(* IEC 61131-3 sources: elnaProjects/ElpcLogic/PomarKc7Changed/build_USO_ecl/_ (part 2) *)

  AI_Tstali_statora_kanal_1_HL := ai.Tstali_statora_kanal_1.HL;
  AI_Tstali_statora_kanal_1_LL := ai.Tstali_statora_kanal_1.LL;
  AI_Tstali_statora_kanal_1_status := DWORD_TO_UDINT(ai.Tstali_statora_kanal_1.status);
  AI_Tstali_statora_kanal_1_value := ai.Tstali_statora_kanal_1.value;
  AI_Tstali_statora_kanal_1_HW := ai.Tstali_statora_kanal_1.HW;
  AI_Tstali_statora_kanal_1_newHW := ai.Tstali_statora_kanal_1.dHW;

  AI_Tstali_statora_kanal_2_HL := ai.Tstali_statora_kanal_2.HL;
  AI_Tstali_statora_kanal_2_LL := ai.Tstali_statora_kanal_2.LL;
  AI_Tstali_statora_kanal_2_status := DWORD_TO_UDINT(ai.Tstali_statora_kanal_2.status);
  AI_Tstali_statora_kanal_2_value := ai.Tstali_statora_kanal_2.value;
  AI_Tstali_statora_kanal_2_HW := ai.Tstali_statora_kanal_2.HW;
  AI_Tstali_statora_kanal_2_newHW := ai.Tstali_statora_kanal_2.dHW;

  AI_Tstali_statora_kanal_3_HL := ai.Tstali_statora_kanal_3.HL;
  AI_Tstali_statora_kanal_3_LL := ai.Tstali_statora_kanal_3.LL;
  AI_Tstali_statora_kanal_3_status := DWORD_TO_UDINT(ai.Tstali_statora_kanal_3.status);
  AI_Tstali_statora_kanal_3_value := ai.Tstali_statora_kanal_3.value;
  AI_Tstali_statora_kanal_3_HW := ai.Tstali_statora_kanal_3.HW;
  AI_Tstali_statora_kanal_3_newHW := ai.Tstali_statora_kanal_3.dHW;

  AI_Tmedi_statora_kanal_1_HL := ai.Tmedi_statora_kanal_1.HL;
  AI_Tmedi_statora_kanal_1_LL := ai.Tmedi_statora_kanal_1.LL;
  AI_Tmedi_statora_kanal_1_status := DWORD_TO_UDINT(ai.Tmedi_statora_kanal_1.status);
  AI_Tmedi_statora_kanal_1_value := ai.Tmedi_statora_kanal_1.value;
  AI_Tmedi_statora_kanal_1_HW := ai.Tmedi_statora_kanal_1.HW;
  AI_Tmedi_statora_kanal_1_newHW := ai.Tmedi_statora_kanal_1.dHW;

  AI_Tmedi_statora_kanal_2_HL := ai.Tmedi_statora_kanal_2.HL;
  AI_Tmedi_statora_kanal_2_LL := ai.Tmedi_statora_kanal_2.LL;
  AI_Tmedi_statora_kanal_2_status := DWORD_TO_UDINT(ai.Tmedi_statora_kanal_2.status);
  AI_Tmedi_statora_kanal_2_value := ai.Tmedi_statora_kanal_2.value;
  AI_Tmedi_statora_kanal_2_HW := ai.Tmedi_statora_kanal_2.HW;
  AI_Tmedi_statora_kanal_2_newHW := ai.Tmedi_statora_kanal_2.dHW;

  AI_Tmedi_statora_kanal_3_HL := ai.Tmedi_statora_kanal_3.HL;
  AI_Tmedi_statora_kanal_3_LL := ai.Tmedi_statora_kanal_3.LL;
  AI_Tmedi_statora_kanal_3_status := DWORD_TO_UDINT(ai.Tmedi_statora_kanal_3.status);
  AI_Tmedi_statora_kanal_3_value := ai.Tmedi_statora_kanal_3.value;
  AI_Tmedi_statora_kanal_3_HW := ai.Tmedi_statora_kanal_3.HW;
  AI_Tmedi_statora_kanal_3_newHW := ai.Tmedi_statora_kanal_3.dHW;

  AI_Toporno_podshipnika_EDT_1_HL := ai.Toporno_podshipnika_EDT_1.HL;
  AI_Toporno_podshipnika_EDT_1_LL := ai.Toporno_podshipnika_EDT_1.LL;
  AI_Toporno_podshipnika_EDT_1_status := DWORD_TO_UDINT(ai.Toporno_podshipnika_EDT_1.status);
  AI_Toporno_podshipnika_EDT_1_value := ai.Toporno_podshipnika_EDT_1.value;
  AI_Toporno_podshipnika_EDT_1_HW := ai.Toporno_podshipnika_EDT_1.HW;
  AI_Toporno_podshipnika_EDT_1_newHW := ai.Toporno_podshipnika_EDT_1.dHW;
  AI_Toporno_podshipnika_EDT_1_HA := ai.Toporno_podshipnika_EDT_1.HA;
  AI_Toporno_podshipnika_EDT_1_newHA := ai.Toporno_podshipnika_EDT_1.dHA;

  AI_Toy_podshipnika_EDT_2_HL := ai.Toy_podshipnika_EDT_2.HL;
  AI_Toy_podshipnika_EDT_2_LL := ai.Toy_podshipnika_EDT_2.LL;
  AI_Toy_podshipnika_EDT_2_status := DWORD_TO_UDINT(ai.Toy_podshipnika_EDT_2.status);
  AI_Toy_podshipnika_EDT_2_value := ai.Toy_podshipnika_EDT_2.value;
  AI_Toy_podshipnika_EDT_2_HW := ai.Toy_podshipnika_EDT_2.HW;
  AI_Toy_podshipnika_EDT_2_newHW := ai.Toy_podshipnika_EDT_2.dHW;
  AI_Toy_podshipnika_EDT_2_HA := ai.Toy_podshipnika_EDT_2.HA;
  AI_Toy_podshipnika_EDT_2_newHA := ai.Toy_podshipnika_EDT_2.dHA;

  AI_Toy_podshipnika_kol_EDT_3_HL := ai.Toy_podshipnika_kol_EDT_3.HL;
  AI_Toy_podshipnika_kol_EDT_3_LL := ai.Toy_podshipnika_kol_EDT_3.LL;
  AI_Toy_podshipnika_kol_EDT_3_status := DWORD_TO_UDINT(ai.Toy_podshipnika_kol_EDT_3.status);
  AI_Toy_podshipnika_kol_EDT_3_value := ai.Toy_podshipnika_kol_EDT_3.value;
  AI_Toy_podshipnika_kol_EDT_3_HW := ai.Toy_podshipnika_kol_EDT_3.HW;
  AI_Toy_podshipnika_kol_EDT_3_newHW := ai.Toy_podshipnika_kol_EDT_3.dHW;
  AI_Toy_podshipnika_kol_EDT_3_HA := ai.Toy_podshipnika_kol_EDT_3.HA;
  AI_Toy_podshipnika_kol_EDT_3_newHA := ai.Toy_podshipnika_kol_EDT_3.dHA;

  AI_Toy_podshipnika_kol_EDT_4_HL := ai.Toy_podshipnika_kol_EDT_4.HL;
  AI_Toy_podshipnika_kol_EDT_4_LL := ai.Toy_podshipnika_kol_EDT_4.LL;
  AI_Toy_podshipnika_kol_EDT_4_status := DWORD_TO_UDINT(ai.Toy_podshipnika_kol_EDT_4.status);
  AI_Toy_podshipnika_kol_EDT_4_value := ai.Toy_podshipnika_kol_EDT_4.value;
  AI_Toy_podshipnika_kol_EDT_4_HW := ai.Toy_podshipnika_kol_EDT_4.HW;
  AI_Toy_podshipnika_kol_EDT_4_newHW := ai.Toy_podshipnika_kol_EDT_4.dHW;
  AI_Toy_podshipnika_kol_EDT_4_HA := ai.Toy_podshipnika_kol_EDT_4.HA;
  AI_Toy_podshipnika_kol_EDT_4_newHA := ai.Toy_podshipnika_kol_EDT_4.dHA;

  AI_Toy_podshipnika_shest_red_EDT_5_HL := ai.Toy_podshipnika_shest_red_EDT_5.HL;
  AI_Toy_podshipnika_shest_red_EDT_5_LL := ai.Toy_podshipnika_shest_red_EDT_5.LL;
  AI_Toy_podshipnika_shest_red_EDT_5_status := DWORD_TO_UDINT(ai.Toy_podshipnika_shest_red_EDT_5.status);
  AI_Toy_podshipnika_shest_red_EDT_5_value := ai.Toy_podshipnika_shest_red_EDT_5.value;
  AI_Toy_podshipnika_shest_red_EDT_5_HW := ai.Toy_podshipnika_shest_red_EDT_5.HW;
  AI_Toy_podshipnika_shest_red_EDT_5_newHW := ai.Toy_podshipnika_shest_red_EDT_5.dHW;
  AI_Toy_podshipnika_shest_red_EDT_5_HA := ai.Toy_podshipnika_shest_red_EDT_5.HA;
  AI_Toy_podshipnika_shest_red_EDT_5_newHA := ai.Toy_podshipnika_shest_red_EDT_5.dHA;

  AI_Ty_podshipnika_red_EDT_6_HL := ai.Ty_podshipnika_red_EDT_6.HL;
  AI_Ty_podshipnika_red_EDT_6_LL := ai.Ty_podshipnika_red_EDT_6.LL;
  AI_Ty_podshipnika_red_EDT_6_status := DWORD_TO_UDINT(ai.Ty_podshipnika_red_EDT_6.status);
  AI_Ty_podshipnika_red_EDT_6_value := ai.Ty_podshipnika_red_EDT_6.value;
  AI_Ty_podshipnika_red_EDT_6_HW := ai.Ty_podshipnika_red_EDT_6.HW;
  AI_Ty_podshipnika_red_EDT_6_newHW := ai.Ty_podshipnika_red_EDT_6.dHW;
  AI_Ty_podshipnika_red_EDT_6_HA := ai.Ty_podshipnika_red_EDT_6.HA;
  AI_Ty_podshipnika_red_EDT_6_newHA := ai.Ty_podshipnika_red_EDT_6.dHA;

  AI_Ty_podshipnika_nagnet_EDT_7_1_HL := ai.Ty_podshipnika_nagnet_EDT_7_1.HL;
  AI_Ty_podshipnika_nagnet_EDT_7_1_LL := ai.Ty_podshipnika_nagnet_EDT_7_1.LL;
  AI_Ty_podshipnika_nagnet_EDT_7_1_status := DWORD_TO_UDINT(ai.Ty_podshipnika_nagnet_EDT_7_1.status);
  AI_Ty_podshipnika_nagnet_EDT_7_1_value := ai.Ty_podshipnika_nagnet_EDT_7_1.value;
  AI_Ty_podshipnika_nagnet_EDT_7_1_HW := ai.Ty_podshipnika_nagnet_EDT_7_1.HW;
  AI_Ty_podshipnika_nagnet_EDT_7_1_newHW := ai.Ty_podshipnika_nagnet_EDT_7_1.dHW;
  AI_Ty_podshipnika_nagnet_EDT_7_1_HA := ai.Ty_podshipnika_nagnet_EDT_7_1.HA;
  AI_Ty_podshipnika_nagnet_EDT_7_1_newHA := ai.Ty_podshipnika_nagnet_EDT_7_1.dHA;

  AI_Ty_podshipnika_nagnet_EDT_7_2_HL := ai.Ty_podshipnika_nagnet_EDT_7_2.HL;
  AI_Ty_podshipnika_nagnet_EDT_7_2_LL := ai.Ty_podshipnika_nagnet_EDT_7_2.LL;
  AI_Ty_podshipnika_nagnet_EDT_7_2_status := DWORD_TO_UDINT(ai.Ty_podshipnika_nagnet_EDT_7_2.status);
  AI_Ty_podshipnika_nagnet_EDT_7_2_value := ai.Ty_podshipnika_nagnet_EDT_7_2.value;
  AI_Ty_podshipnika_nagnet_EDT_7_2_HW := ai.Ty_podshipnika_nagnet_EDT_7_2.HW;
  AI_Ty_podshipnika_nagnet_EDT_7_2_newHW := ai.Ty_podshipnika_nagnet_EDT_7_2.dHW;
  AI_Ty_podshipnika_nagnet_EDT_7_2_HA := ai.Ty_podshipnika_nagnet_EDT_7_2.HA;
  AI_Ty_podshipnika_nagnet_EDT_7_2_newHA := ai.Ty_podshipnika_nagnet_EDT_7_2.dHA;

  AI_Toy_podshipnika_svobod_konca_EDT_8_1_HL := ai.Toy_podshipnika_svobod_konca_EDT_8_1.HL;
  AI_Toy_podshipnika_svobod_konca_EDT_8_1_LL := ai.Toy_podshipnika_svobod_konca_EDT_8_1.LL;
  AI_Toy_podshipnika_svobod_konca_EDT_8_1_status := DWORD_TO_UDINT(ai.Toy_podshipnika_svobod_konca_EDT_8_1.status);
  AI_Toy_podshipnika_svobod_konca_EDT_8_1_value := ai.Toy_podshipnika_svobod_konca_EDT_8_1.value;
  AI_Toy_podshipnika_svobod_konca_EDT_8_1_HW := ai.Toy_podshipnika_svobod_konca_EDT_8_1.HW;
  AI_Toy_podshipnika_svobod_konca_EDT_8_1_newHW := ai.Toy_podshipnika_svobod_konca_EDT_8_1.dHW;
  AI_Toy_podshipnika_svobod_konca_EDT_8_1_HA := ai.Toy_podshipnika_svobod_konca_EDT_8_1.HA;
  AI_Toy_podshipnika_svobod_konca_EDT_8_1_newHA := ai.Toy_podshipnika_svobod_konca_EDT_8_1.dHA;

  AI_Toy_podshipnika_svobod_konca_EDT_8_2_HL := ai.Toy_podshipnika_svobod_konca_EDT_8_2.HL;
  AI_Toy_podshipnika_svobod_konca_EDT_8_2_LL := ai.Toy_podshipnika_svobod_konca_EDT_8_2.LL;
  AI_Toy_podshipnika_svobod_konca_EDT_8_2_status := DWORD_TO_UDINT(ai.Toy_podshipnika_svobod_konca_EDT_8_2.status);
  AI_Toy_podshipnika_svobod_konca_EDT_8_2_value := ai.Toy_podshipnika_svobod_konca_EDT_8_2.value;
  AI_Toy_podshipnika_svobod_konca_EDT_8_2_HW := ai.Toy_podshipnika_svobod_konca_EDT_8_2.HW;
  AI_Toy_podshipnika_svobod_konca_EDT_8_2_newHW := ai.Toy_podshipnika_svobod_konca_EDT_8_2.dHW;
  AI_Toy_podshipnika_svobod_konca_EDT_8_2_HA := ai.Toy_podshipnika_svobod_konca_EDT_8_2.HA;
  AI_Toy_podshipnika_svobod_konca_EDT_8_2_newHA := ai.Toy_podshipnika_svobod_konca_EDT_8_2.dHA;

  AI_Toy_podshipnika_rab_kol_EDT_9_1_HL := ai.Toy_podshipnika_rab_kol_EDT_9_1.HL;
  AI_Toy_podshipnika_rab_kol_EDT_9_1_LL := ai.Toy_podshipnika_rab_kol_EDT_9_1.LL;
  AI_Toy_podshipnika_rab_kol_EDT_9_1_status := DWORD_TO_UDINT(ai.Toy_podshipnika_rab_kol_EDT_9_1.status);
  AI_Toy_podshipnika_rab_kol_EDT_9_1_value := ai.Toy_podshipnika_rab_kol_EDT_9_1.value;
  AI_Toy_podshipnika_rab_kol_EDT_9_1_HW := ai.Toy_podshipnika_rab_kol_EDT_9_1.HW;
  AI_Toy_podshipnika_rab_kol_EDT_9_1_newHW := ai.Toy_podshipnika_rab_kol_EDT_9_1.dHW;
  AI_Toy_podshipnika_rab_kol_EDT_9_1_HA := ai.Toy_podshipnika_rab_kol_EDT_9_1.HA;
  AI_Toy_podshipnika_rab_kol_EDT_9_1_newHA := ai.Toy_podshipnika_rab_kol_EDT_9_1.dHA;

  AI_Toy_podshipnika_rab_kol_EDT_9_2_HL := ai.Toy_podshipnika_rab_kol_EDT_9_2.HL;
  AI_Toy_podshipnika_rab_kol_EDT_9_2_LL := ai.Toy_podshipnika_rab_kol_EDT_9_2.LL;
  AI_Toy_podshipnika_rab_kol_EDT_9_2_status := DWORD_TO_UDINT(ai.Toy_podshipnika_rab_kol_EDT_9_2.status);
  AI_Toy_podshipnika_rab_kol_EDT_9_2_value := ai.Toy_podshipnika_rab_kol_EDT_9_2.value;
  AI_Toy_podshipnika_rab_kol_EDT_9_2_HW := ai.Toy_podshipnika_rab_kol_EDT_9_2.HW;
  AI_Toy_podshipnika_rab_kol_EDT_9_2_newHW := ai.Toy_podshipnika_rab_kol_EDT_9_2.dHW;
  AI_Toy_podshipnika_rab_kol_EDT_9_2_HA := ai.Toy_podshipnika_rab_kol_EDT_9_2.HA;
  AI_Toy_podshipnika_rab_kol_EDT_9_2_newHA := ai.Toy_podshipnika_rab_kol_EDT_9_2.dHA;

  AI_Toy_podshipnika_nerab_kol_EDT_10_1_HL := ai.Toy_podshipnika_nerab_kol_EDT_10_1.HL;
  AI_Toy_podshipnika_nerab_kol_EDT_10_1_LL := ai.Toy_podshipnika_nerab_kol_EDT_10_1.LL;
  AI_Toy_podshipnika_nerab_kol_EDT_10_1_status := DWORD_TO_UDINT(ai.Toy_podshipnika_nerab_kol_EDT_10_1.status);
  AI_Toy_podshipnika_nerab_kol_EDT_10_1_value := ai.Toy_podshipnika_nerab_kol_EDT_10_1.value;
  AI_Toy_podshipnika_nerab_kol_EDT_10_1_HW := ai.Toy_podshipnika_nerab_kol_EDT_10_1.HW;
  AI_Toy_podshipnika_nerab_kol_EDT_10_1_newHW := ai.Toy_podshipnika_nerab_kol_EDT_10_1.dHW;
  AI_Toy_podshipnika_nerab_kol_EDT_10_1_HA := ai.Toy_podshipnika_nerab_kol_EDT_10_1.HA;
  AI_Toy_podshipnika_nerab_kol_EDT_10_1_newHA := ai.Toy_podshipnika_nerab_kol_EDT_10_1.dHA;

  AI_Toy_podshipnika_nerab_kol_EDT_10_2_HL := ai.Toy_podshipnika_nerab_kol_EDT_10_2.HL;
  AI_Toy_podshipnika_nerab_kol_EDT_10_2_LL := ai.Toy_podshipnika_nerab_kol_EDT_10_2.LL;
  AI_Toy_podshipnika_nerab_kol_EDT_10_2_status := DWORD_TO_UDINT(ai.Toy_podshipnika_nerab_kol_EDT_10_2.status);
  AI_Toy_podshipnika_nerab_kol_EDT_10_2_value := ai.Toy_podshipnika_nerab_kol_EDT_10_2.value;
  AI_Toy_podshipnika_nerab_kol_EDT_10_2_HW := ai.Toy_podshipnika_nerab_kol_EDT_10_2.HW;
  AI_Toy_podshipnika_nerab_kol_EDT_10_2_newHW := ai.Toy_podshipnika_nerab_kol_EDT_10_2.dHW;
  AI_Toy_podshipnika_nerab_kol_EDT_10_2_HA := ai.Toy_podshipnika_nerab_kol_EDT_10_2.HA;
  AI_Toy_podshipnika_nerab_kol_EDT_10_2_newHA := ai.Toy_podshipnika_nerab_kol_EDT_10_2.dHA;

  AI_Tholodnogo_vozduha_ED_kanal_1_HL := ai.Tholodnogo_vozduha_ED_kanal_1.HL;
  AI_Tholodnogo_vozduha_ED_kanal_1_LL := ai.Tholodnogo_vozduha_ED_kanal_1.LL;
  AI_Tholodnogo_vozduha_ED_kanal_1_status := DWORD_TO_UDINT(ai.Tholodnogo_vozduha_ED_kanal_1.status);
  AI_Tholodnogo_vozduha_ED_kanal_1_value := ai.Tholodnogo_vozduha_ED_kanal_1.value;
  AI_Tholodnogo_vozduha_ED_kanal_1_HW := ai.Tholodnogo_vozduha_ED_kanal_1.HW;
  AI_Tholodnogo_vozduha_ED_kanal_1_newHW := ai.Tholodnogo_vozduha_ED_kanal_1.dHW;

  AI_Tholodnogo_vozduha_ED_kanal_2_HL := ai.Tholodnogo_vozduha_ED_kanal_2.HL;
  AI_Tholodnogo_vozduha_ED_kanal_2_LL := ai.Tholodnogo_vozduha_ED_kanal_2.LL;
  AI_Tholodnogo_vozduha_ED_kanal_2_status := DWORD_TO_UDINT(ai.Tholodnogo_vozduha_ED_kanal_2.status);
  AI_Tholodnogo_vozduha_ED_kanal_2_value := ai.Tholodnogo_vozduha_ED_kanal_2.value;
  AI_Tholodnogo_vozduha_ED_kanal_2_HW := ai.Tholodnogo_vozduha_ED_kanal_2.HW;
  AI_Tholodnogo_vozduha_ED_kanal_2_newHW := ai.Tholodnogo_vozduha_ED_kanal_2.dHW;

  AI_Tgorjachego_vozduha_ED_kanal_1_HL := ai.Tgorjachego_vozduha_ED_kanal_1.HL;
  AI_Tgorjachego_vozduha_ED_kanal_1_LL := ai.Tgorjachego_vozduha_ED_kanal_1.LL;
  AI_Tgorjachego_vozduha_ED_kanal_1_status := DWORD_TO_UDINT(ai.Tgorjachego_vozduha_ED_kanal_1.status);
  AI_Tgorjachego_vozduha_ED_kanal_1_value := ai.Tgorjachego_vozduha_ED_kanal_1.value;
  AI_Tgorjachego_vozduha_ED_kanal_1_HW := ai.Tgorjachego_vozduha_ED_kanal_1.HW;
  AI_Tgorjachego_vozduha_ED_kanal_1_newHW := ai.Tgorjachego_vozduha_ED_kanal_1.dHW;

  AI_Tgorjachego_vozduha_ED_kanal_2_HL := ai.Tgorjachego_vozduha_ED_kanal_2.HL;
  AI_Tgorjachego_vozduha_ED_kanal_2_LL := ai.Tgorjachego_vozduha_ED_kanal_2.LL;
  AI_Tgorjachego_vozduha_ED_kanal_2_status := DWORD_TO_UDINT(ai.Tgorjachego_vozduha_ED_kanal_2.status);
  AI_Tgorjachego_vozduha_ED_kanal_2_value := ai.Tgorjachego_vozduha_ED_kanal_2.value;
  AI_Tgorjachego_vozduha_ED_kanal_2_HW := ai.Tgorjachego_vozduha_ED_kanal_2.HW;
  AI_Tgorjachego_vozduha_ED_kanal_2_newHW := ai.Tgorjachego_vozduha_ED_kanal_2.dHW;

  AI_Tnarujnogo_vozduha_HL := ai.Tnarujnogo_vozduha.HL;
  AI_Tnarujnogo_vozduha_LL := ai.Tnarujnogo_vozduha.LL;
  AI_Tnarujnogo_vozduha_status := DWORD_TO_UDINT(ai.Tnarujnogo_vozduha.status);
  AI_Tnarujnogo_vozduha_value := ai.Tnarujnogo_vozduha.value;
  AI_Tnarujnogo_vozduha_HW := ai.Tnarujnogo_vozduha.HW;
  AI_Tnarujnogo_vozduha_newHW := ai.Tnarujnogo_vozduha.dHW;

  AI_Tgaza_na_vhode_H_HL := ai.Tgaza_na_vhode_H.HL;
  AI_Tgaza_na_vhode_H_LL := ai.Tgaza_na_vhode_H.LL;
  AI_Tgaza_na_vhode_H_status := DWORD_TO_UDINT(ai.Tgaza_na_vhode_H.status);
  AI_Tgaza_na_vhode_H_value := ai.Tgaza_na_vhode_H.value;
  AI_Tgaza_na_vhode_H_HW := ai.Tgaza_na_vhode_H.HW;
  AI_Tgaza_na_vhode_H_newHW := ai.Tgaza_na_vhode_H.dHW;

  AI_Tgaza_na_vyhode_H_HL := ai.Tgaza_na_vyhode_H.HL;
  AI_Tgaza_na_vyhode_H_LL := ai.Tgaza_na_vyhode_H.LL;
  AI_Tgaza_na_vyhode_H_status := DWORD_TO_UDINT(ai.Tgaza_na_vyhode_H.status);
  AI_Tgaza_na_vyhode_H_value := ai.Tgaza_na_vyhode_H.value;
  AI_Tgaza_na_vyhode_H_HW := ai.Tgaza_na_vyhode_H.HW;
  AI_Tgaza_na_vyhode_H_newHW := ai.Tgaza_na_vyhode_H.dHW;
  AI_Tgaza_na_vyhode_H_HA := ai.Tgaza_na_vyhode_H.HA;
  AI_Tgaza_na_vyhode_H_newHA := ai.Tgaza_na_vyhode_H.dHA;

  AI_Tmasla_do_AVOM_HL := ai.Tmasla_do_AVOM.HL;
  AI_Tmasla_do_AVOM_LL := ai.Tmasla_do_AVOM.LL;
  AI_Tmasla_do_AVOM_status := DWORD_TO_UDINT(ai.Tmasla_do_AVOM.status);
  AI_Tmasla_do_AVOM_value := ai.Tmasla_do_AVOM.value;
  AI_Tmasla_do_AVOM_HW := ai.Tmasla_do_AVOM.HW;
  AI_Tmasla_do_AVOM_newHW := ai.Tmasla_do_AVOM.dHW;

  AI_Tmasla_posle_AVOM_HL := ai.Tmasla_posle_AVOM.HL;
  AI_Tmasla_posle_AVOM_LL := ai.Tmasla_posle_AVOM.LL;
  AI_Tmasla_posle_AVOM_status := DWORD_TO_UDINT(ai.Tmasla_posle_AVOM.status);
  AI_Tmasla_posle_AVOM_value := ai.Tmasla_posle_AVOM.value;
  AI_Tmasla_posle_AVOM_HW := ai.Tmasla_posle_AVOM.HW;
  AI_Tmasla_posle_AVOM_newHW := ai.Tmasla_posle_AVOM.dHW;

  AI_Tmasla_MB_HL := ai.Tmasla_MB.HL;
  AI_Tmasla_MB_LL := ai.Tmasla_MB.LL;
  AI_Tmasla_MB_status := DWORD_TO_UDINT(ai.Tmasla_MB.status);
  AI_Tmasla_MB_value := ai.Tmasla_MB.value;
  AI_Tmasla_MB_LW := ai.Tmasla_MB.LW;
  AI_Tmasla_MB_newLW := ai.Tmasla_MB.dLW;

  AI_Tmasla_MB_TEN_HL := ai.Tmasla_MB_TEN.HL;
  AI_Tmasla_MB_TEN_LL := ai.Tmasla_MB_TEN.LL;
  AI_Tmasla_MB_TEN_status := DWORD_TO_UDINT(ai.Tmasla_MB_TEN.status);
  AI_Tmasla_MB_TEN_value := ai.Tmasla_MB_TEN.value;
  AI_Tmasla_MB_TEN_HW := ai.Tmasla_MB_TEN.HW;
  AI_Tmasla_MB_TEN_newHW := ai.Tmasla_MB_TEN.dHW;

  AI_Tshu_HL := ai.Tshu.HL;
  AI_Tshu_LL := ai.Tshu.LL;
  AI_Tshu_status := DWORD_TO_UDINT(ai.Tshu.status);
  AI_Tshu_value := ai.Tshu.value;

  AI_Pmaslo_sm_nizkoe_HL := ai.Pmaslo_sm_nizkoe.HL;
  AI_Pmaslo_sm_nizkoe_LL := ai.Pmaslo_sm_nizkoe.LL;
  AI_Pmaslo_sm_nizkoe_status := DWORD_TO_UDINT(ai.Pmaslo_sm_nizkoe.status);
  AI_Pmaslo_sm_nizkoe_value := ai.Pmaslo_sm_nizkoe.value;
  AI_Pmaslo_sm_nizkoe_LW := ai.Pmaslo_sm_nizkoe.LW;
  AI_Pmaslo_sm_nizkoe_newLW := ai.Pmaslo_sm_nizkoe.dLW;
  AI_Pmaslo_sm_nizkoe_LA := ai.Pmaslo_sm_nizkoe.LA;
  AI_Pmaslo_sm_nizkoe_newLA := ai.Pmaslo_sm_nizkoe.dLA;

  AI_Pmaslo_sm_vysokoe_HL := ai.Pmaslo_sm_vysokoe.HL;
  AI_Pmaslo_sm_vysokoe_LL := ai.Pmaslo_sm_vysokoe.LL;
  AI_Pmaslo_sm_vysokoe_status := DWORD_TO_UDINT(ai.Pmaslo_sm_vysokoe.status);
  AI_Pmaslo_sm_vysokoe_value := ai.Pmaslo_sm_vysokoe.value;
  AI_Pmaslo_sm_vysokoe_LW := ai.Pmaslo_sm_vysokoe.LW;
  AI_Pmaslo_sm_vysokoe_newLW := ai.Pmaslo_sm_vysokoe.dLW;
  AI_Pmaslo_sm_vysokoe_LA := ai.Pmaslo_sm_vysokoe.LA;
  AI_Pmaslo_sm_vysokoe_newLA := ai.Pmaslo_sm_vysokoe.dLA;

  AI_Pmasla_posle_GNS_HL := ai.Pmasla_posle_GNS.HL;
  AI_Pmasla_posle_GNS_LL := ai.Pmasla_posle_GNS.LL;
  AI_Pmasla_posle_GNS_status := DWORD_TO_UDINT(ai.Pmasla_posle_GNS.status);
  AI_Pmasla_posle_GNS_value := ai.Pmasla_posle_GNS.value;
  AI_Pmasla_posle_GNS_HW := ai.Pmasla_posle_GNS.HW;
  AI_Pmasla_posle_GNS_newHW := ai.Pmasla_posle_GNS.dHW;
  AI_Pmasla_posle_GNS_LW := ai.Pmasla_posle_GNS.LW;
  AI_Pmasla_posle_GNS_newLW := ai.Pmasla_posle_GNS.dLW;

  AI_Pmasla_posle_NU_HL := ai.Pmasla_posle_NU.HL;
  AI_Pmasla_posle_NU_LL := ai.Pmasla_posle_NU.LL;
  AI_Pmasla_posle_NU_status := DWORD_TO_UDINT(ai.Pmasla_posle_NU.status);
  AI_Pmasla_posle_NU_value := ai.Pmasla_posle_NU.value;
  AI_Pmasla_posle_NU_LW := ai.Pmasla_posle_NU.LW;
  AI_Pmasla_posle_NU_newLW := ai.Pmasla_posle_NU.dLW;

  AI_Pgaza_na_vhode_nagnetatelia_HL := ai.Pgaza_na_vhode_nagnetatelia.HL;
  AI_Pgaza_na_vhode_nagnetatelia_LL := ai.Pgaza_na_vhode_nagnetatelia.LL;
  AI_Pgaza_na_vhode_nagnetatelia_status := DWORD_TO_UDINT(ai.Pgaza_na_vhode_nagnetatelia.status);
  AI_Pgaza_na_vhode_nagnetatelia_value := ai.Pgaza_na_vhode_nagnetatelia.value;
  AI_Pgaza_na_vhode_nagnetatelia_LW := ai.Pgaza_na_vhode_nagnetatelia.LW;
  AI_Pgaza_na_vhode_nagnetatelia_newLW := ai.Pgaza_na_vhode_nagnetatelia.dLW;

  AI_Pgaza_na_vyhode_nagnetatelia_HL := ai.Pgaza_na_vyhode_nagnetatelia.HL;
  AI_Pgaza_na_vyhode_nagnetatelia_LL := ai.Pgaza_na_vyhode_nagnetatelia.LL;
  AI_Pgaza_na_vyhode_nagnetatelia_status := DWORD_TO_UDINT(ai.Pgaza_na_vyhode_nagnetatelia.status);
  AI_Pgaza_na_vyhode_nagnetatelia_value := ai.Pgaza_na_vyhode_nagnetatelia.value;
  AI_Pgaza_na_vyhode_nagnetatelia_HW := ai.Pgaza_na_vyhode_nagnetatelia.HW;
  AI_Pgaza_na_vyhode_nagnetatelia_newHW := ai.Pgaza_na_vyhode_nagnetatelia.dHW;
  AI_Pgaza_na_vyhode_nagnetatelia_HA := ai.Pgaza_na_vyhode_nagnetatelia.HA;
  AI_Pgaza_na_vyhode_nagnetatelia_newHA := ai.Pgaza_na_vyhode_nagnetatelia.dHA;

  AI_Pimpuls_gaz_HL := ai.Pimpuls_gaz.HL;
  AI_Pimpuls_gaz_LL := ai.Pimpuls_gaz.LL;
  AI_Pimpuls_gaz_status := DWORD_TO_UDINT(ai.Pimpuls_gaz.status);
  AI_Pimpuls_gaz_value := ai.Pimpuls_gaz.value;
  AI_Pimpuls_gaz_LW := ai.Pimpuls_gaz.LW;
  AI_Pimpuls_gaz_newLW := ai.Pimpuls_gaz.dLW;

  AI_dPgaza_na_maslo_filtre_HL := ai.dPgaza_na_maslo_filtre.HL;
  AI_dPgaza_na_maslo_filtre_LL := ai.dPgaza_na_maslo_filtre.LL;
  AI_dPgaza_na_maslo_filtre_status := DWORD_TO_UDINT(ai.dPgaza_na_maslo_filtre.status);
  AI_dPgaza_na_maslo_filtre_value := ai.dPgaza_na_maslo_filtre.value;
  AI_dPgaza_na_maslo_filtre_HW := ai.dPgaza_na_maslo_filtre.HW;
  AI_dPgaza_na_maslo_filtre_newHW := ai.dPgaza_na_maslo_filtre.dHW;

  AI_dPgaza_na_konfuzore_HL := ai.dPgaza_na_konfuzore.HL;
  AI_dPgaza_na_konfuzore_LL := ai.dPgaza_na_konfuzore.LL;
  AI_dPgaza_na_konfuzore_status := DWORD_TO_UDINT(ai.dPgaza_na_konfuzore.status);
  AI_dPgaza_na_konfuzore_value := ai.dPgaza_na_konfuzore.value;
  AI_dPgaza_na_konfuzore_LW := ai.dPgaza_na_konfuzore.LW;
  AI_dPgaza_na_konfuzore_newLW := ai.dPgaza_na_konfuzore.dLW;

  AI_dPmaslo_gaz_HL := ai.dPmaslo_gaz.HL;
  AI_dPmaslo_gaz_LL := ai.dPmaslo_gaz.LL;
  AI_dPmaslo_gaz_status := DWORD_TO_UDINT(ai.dPmaslo_gaz.status);
  AI_dPmaslo_gaz_value := ai.dPmaslo_gaz.value;
  AI_dPmaslo_gaz_LW := ai.dPmaslo_gaz.LW;
  AI_dPmaslo_gaz_newLW := ai.dPmaslo_gaz.dLW;
  AI_dPmaslo_gaz_LA := ai.dPmaslo_gaz.LA;
  AI_dPmaslo_gaz_newLA := ai.dPmaslo_gaz.dLA;

  AI_Os_sdvig_nagnetatelja_plus_HL := ai.Os_sdvig_nagnetatelja_plus.HL;
  AI_Os_sdvig_nagnetatelja_plus_LL := ai.Os_sdvig_nagnetatelja_plus.LL;
  AI_Os_sdvig_nagnetatelja_plus_status := DWORD_TO_UDINT(ai.Os_sdvig_nagnetatelja_plus.status);
  AI_Os_sdvig_nagnetatelja_plus_value := ai.Os_sdvig_nagnetatelja_plus.value;
  AI_Os_sdvig_nagnetatelja_plus_HW := ai.Os_sdvig_nagnetatelja_plus.HW;
  AI_Os_sdvig_nagnetatelja_plus_newHW := ai.Os_sdvig_nagnetatelja_plus.dHW;
  AI_Os_sdvig_nagnetatelja_plus_HA := ai.Os_sdvig_nagnetatelja_plus.HA;
  AI_Os_sdvig_nagnetatelja_plus_newHA := ai.Os_sdvig_nagnetatelja_plus.dHA;

  AI_Os_sdvig_nagnetatelja_minus_HL := ai.Os_sdvig_nagnetatelja_minus.HL;
  AI_Os_sdvig_nagnetatelja_minus_LL := ai.Os_sdvig_nagnetatelja_minus.LL;
  AI_Os_sdvig_nagnetatelja_minus_status := DWORD_TO_UDINT(ai.Os_sdvig_nagnetatelja_minus.status);
  AI_Os_sdvig_nagnetatelja_minus_value := ai.Os_sdvig_nagnetatelja_minus.value;
  AI_Os_sdvig_nagnetatelja_minus_LW := ai.Os_sdvig_nagnetatelja_minus.LW;
  AI_Os_sdvig_nagnetatelja_minus_newLW := ai.Os_sdvig_nagnetatelja_minus.dLW;
  AI_Os_sdvig_nagnetatelja_minus_LA := ai.Os_sdvig_nagnetatelja_minus.LA;
  AI_Os_sdvig_nagnetatelja_minus_newLA := ai.Os_sdvig_nagnetatelja_minus.dLA;

  AI_Yroven_masla_MB_HL := ai.Yroven_masla_MB.HL;
  AI_Yroven_masla_MB_LL := ai.Yroven_masla_MB.LL;
  AI_Yroven_masla_MB_status := DWORD_TO_UDINT(ai.Yroven_masla_MB.status);
  AI_Yroven_masla_MB_value := ai.Yroven_masla_MB.value;
  AI_Yroven_masla_MB_LW := ai.Yroven_masla_MB.LW;
  AI_Yroven_masla_MB_newLW := ai.Yroven_masla_MB.dLW;

  AI_Kontrol_per_220V_HL := ai.Kontrol_per_220V.HL;
  AI_Kontrol_per_220V_LL := ai.Kontrol_per_220V.LL;
  AI_Kontrol_per_220V_status := DWORD_TO_UDINT(ai.Kontrol_per_220V.status);
  AI_Kontrol_per_220V_value := ai.Kontrol_per_220V.value;
  AI_Kontrol_per_220V_HW := ai.Kontrol_per_220V.HW;
  AI_Kontrol_per_220V_newHW := ai.Kontrol_per_220V.dHW;
  AI_Kontrol_per_220V_LW := ai.Kontrol_per_220V.LW;
  AI_Kontrol_per_220V_newLW := ai.Kontrol_per_220V.dLW;

  AI_Kontrol_post_220V_HL := ai.Kontrol_post_220V.HL;
  AI_Kontrol_post_220V_LL := ai.Kontrol_post_220V.LL;
  AI_Kontrol_post_220V_status := DWORD_TO_UDINT(ai.Kontrol_post_220V.status);
  AI_Kontrol_post_220V_value := ai.Kontrol_post_220V.value;
  AI_Kontrol_post_220V_HW := ai.Kontrol_post_220V.HW;
  AI_Kontrol_post_220V_newHW := ai.Kontrol_post_220V.dHW;
  AI_Kontrol_post_220V_LW := ai.Kontrol_post_220V.LW;
  AI_Kontrol_post_220V_newLW := ai.Kontrol_post_220V.dLW;

  AI_Tok_statora_HL := ai.Tok_statora.HL;
  AI_Tok_statora_LL := ai.Tok_statora.LL;
  AI_Tok_statora_status := DWORD_TO_UDINT(ai.Tok_statora.status);
  AI_Tok_statora_value := ai.Tok_statora.value;
  AI_Tok_statora_LW := ai.Tok_statora.LW;
  AI_Tok_statora_newLW := ai.Tok_statora.dLW;

  AI_Vibro_skorost_OPED_T1_HL := ai.Vibro_skorost_OPED_T1.HL;
  AI_Vibro_skorost_OPED_T1_LL := ai.Vibro_skorost_OPED_T1.LL;
  AI_Vibro_skorost_OPED_T1_status := DWORD_TO_UDINT(ai.Vibro_skorost_OPED_T1.status);
  AI_Vibro_skorost_OPED_T1_value := ai.Vibro_skorost_OPED_T1.value;
  AI_Vibro_skorost_OPED_T1_HW := ai.Vibro_skorost_OPED_T1.HW;
  AI_Vibro_skorost_OPED_T1_newHW := ai.Vibro_skorost_OPED_T1.dHW;
  AI_Vibro_skorost_OPED_T1_HA := ai.Vibro_skorost_OPED_T1.HA;
  AI_Vibro_skorost_OPED_T1_newHA := ai.Vibro_skorost_OPED_T1.dHA;

  AI_Vibro_skorost_OYPED_T2_HL := ai.Vibro_skorost_OYPED_T2.HL;
  AI_Vibro_skorost_OYPED_T2_LL := ai.Vibro_skorost_OYPED_T2.LL;
  AI_Vibro_skorost_OYPED_T2_status := DWORD_TO_UDINT(ai.Vibro_skorost_OYPED_T2.status);
  AI_Vibro_skorost_OYPED_T2_value := ai.Vibro_skorost_OYPED_T2.value;
  AI_Vibro_skorost_OYPED_T2_HW := ai.Vibro_skorost_OYPED_T2.HW;
  AI_Vibro_skorost_OYPED_T2_newHW := ai.Vibro_skorost_OYPED_T2.dHW;
  AI_Vibro_skorost_OYPED_T2_HA := ai.Vibro_skorost_OYPED_T2.HA;
  AI_Vibro_skorost_OYPED_T2_newHA := ai.Vibro_skorost_OYPED_T2.dHA;

  AI_Vibro_skorost_OYP_kolesa_ED_T3_HL := ai.Vibro_skorost_OYP_kolesa_ED_T3.HL;
  AI_Vibro_skorost_OYP_kolesa_ED_T3_LL := ai.Vibro_skorost_OYP_kolesa_ED_T3.LL;
  AI_Vibro_skorost_OYP_kolesa_ED_T3_status := DWORD_TO_UDINT(ai.Vibro_skorost_OYP_kolesa_ED_T3.status);
  AI_Vibro_skorost_OYP_kolesa_ED_T3_value := ai.Vibro_skorost_OYP_kolesa_ED_T3.value;
  AI_Vibro_skorost_OYP_kolesa_ED_T3_HW := ai.Vibro_skorost_OYP_kolesa_ED_T3.HW;
  AI_Vibro_skorost_OYP_kolesa_ED_T3_newHW := ai.Vibro_skorost_OYP_kolesa_ED_T3.dHW;
  AI_Vibro_skorost_OYP_kolesa_ED_T3_HA := ai.Vibro_skorost_OYP_kolesa_ED_T3.HA;
  AI_Vibro_skorost_OYP_kolesa_ED_T3_newHA := ai.Vibro_skorost_OYP_kolesa_ED_T3.dHA;

  AI_Vibro_skorost_OP_kolesa_RH_T4_HL := ai.Vibro_skorost_OP_kolesa_RH_T4.HL;
  AI_Vibro_skorost_OP_kolesa_RH_T4_LL := ai.Vibro_skorost_OP_kolesa_RH_T4.LL;
  AI_Vibro_skorost_OP_kolesa_RH_T4_status := DWORD_TO_UDINT(ai.Vibro_skorost_OP_kolesa_RH_T4.status);
  AI_Vibro_skorost_OP_kolesa_RH_T4_value := ai.Vibro_skorost_OP_kolesa_RH_T4.value;
  AI_Vibro_skorost_OP_kolesa_RH_T4_HW := ai.Vibro_skorost_OP_kolesa_RH_T4.HW;
  AI_Vibro_skorost_OP_kolesa_RH_T4_newHW := ai.Vibro_skorost_OP_kolesa_RH_T4.dHW;
  AI_Vibro_skorost_OP_kolesa_RH_T4_HA := ai.Vibro_skorost_OP_kolesa_RH_T4.HA;
  AI_Vibro_skorost_OP_kolesa_RH_T4_newHA := ai.Vibro_skorost_OP_kolesa_RH_T4.dHA;

  AI_Vibro_skorost_OP_shesterni_RED_T5_HL := ai.Vibro_skorost_OP_shesterni_RED_T5.HL;
  AI_Vibro_skorost_OP_shesterni_RED_T5_LL := ai.Vibro_skorost_OP_shesterni_RED_T5.LL;
  AI_Vibro_skorost_OP_shesterni_RED_T5_status := DWORD_TO_UDINT(ai.Vibro_skorost_OP_shesterni_RED_T5.status);
  AI_Vibro_skorost_OP_shesterni_RED_T5_value := ai.Vibro_skorost_OP_shesterni_RED_T5.value;
  AI_Vibro_skorost_OP_shesterni_RED_T5_HW := ai.Vibro_skorost_OP_shesterni_RED_T5.HW;
  AI_Vibro_skorost_OP_shesterni_RED_T5_newHW := ai.Vibro_skorost_OP_shesterni_RED_T5.dHW;
  AI_Vibro_skorost_OP_shesterni_RED_T5_HA := ai.Vibro_skorost_OP_shesterni_RED_T5.HA;
  AI_Vibro_skorost_OP_shesterni_RED_T5_newHA := ai.Vibro_skorost_OP_shesterni_RED_T5.dHA;

  AI_Vibro_skorost_OP_shesterni_RED_T6_HL := ai.Vibro_skorost_OP_shesterni_RED_T6.HL;
  AI_Vibro_skorost_OP_shesterni_RED_T6_LL := ai.Vibro_skorost_OP_shesterni_RED_T6.LL;
  AI_Vibro_skorost_OP_shesterni_RED_T6_status := DWORD_TO_UDINT(ai.Vibro_skorost_OP_shesterni_RED_T6.status);
  AI_Vibro_skorost_OP_shesterni_RED_T6_value := ai.Vibro_skorost_OP_shesterni_RED_T6.value;
  AI_Vibro_skorost_OP_shesterni_RED_T6_HW := ai.Vibro_skorost_OP_shesterni_RED_T6.HW;
  AI_Vibro_skorost_OP_shesterni_RED_T6_newHW := ai.Vibro_skorost_OP_shesterni_RED_T6.dHW;
  AI_Vibro_skorost_OP_shesterni_RED_T6_HA := ai.Vibro_skorost_OP_shesterni_RED_T6.HA;
  AI_Vibro_skorost_OP_shesterni_RED_T6_newHA := ai.Vibro_skorost_OP_shesterni_RED_T6.dHA;
END_FUNCTION_BLOCK

FUNCTION_BLOCK fb_DualStateIm
  VAR_INPUT
    statOn : BOOL;
    statOff : BOOL;
  END_VAR
  VAR_IN_OUT
    StrDs : struct_DualStateIm;
  END_VAR
  VAR_INPUT
    statOn_reliability : BOOL;
    statOff_reliability : BOOL;
    inNs : TYPE_ReliableBit;
    inAccident : TYPE_ReliableBit;
    inCommand : WORD;
  END_VAR
  VAR
    _statOn : BOOL;
    _statOff : BOOL;
    getSdvig : BOOL;
    lastOnStatus : BYTE;
    cmd : BYTE;
    source : BYTE;
    lastCmd : BYTE;
    source_for_Status : BYTE;
    cmd_for_Status : BYTE;
    command_error_for_Status : BYTE;
    _sunpackerCommand : fb_sunpackerCommand;
    _statusDualInput : TYPE_statusDualInput;
    _commandDualInput : TYPE_commandDualInput;
    _commandErrorTimer : BOOL;
    onInit : BOOL      := FALSE;
    resetErrorTimer : BOOL;
    _changWithoutCommand : BOOL;
    errorCMDTimer : TON;
    sdvigReset : TON;
    _errorReset : TON;
  END_VAR
  VAR_IN_OUT
    cmdOn : BOOL;
  END_VAR
  VAR_OUTPUT
    cmdOff : BOOL;
  END_VAR

  IF NOT onInit THEN
  IF StrDs.ISVALIDREF_cmdOn XOR StrDs.ISVALIDREF_cmdOff THEN
  	IF 	StrDs.ISVALIDREF_cmdOn THEN
  		lastCmd:= 2; (*baseCmdOff*)
  	ELSE
  		lastCmd:= 1; (*baseCmdOn*)
  	END_IF;
  END_IF;
  onInit:=TRUE;
  END_IF;

  (* ---- Если управление с ВУ заблокировано, то в ИМ передаем команду из алгоритма ---- *)
  IF StrDs.inOpcCommandsDisabled THEN
  	StrDs.inCommand := StrDs.inCommand_Alg;
  ELSE (* иначе передаем команду с АРМа*)
  	StrDs.inCommand := StrDs.inCommand_ARM;
  END_IF;

  (* ---- Формирование состояния механизма ---- *)

  IF (StrDs.ISVALIDREF_statOn) OR (StrDs.ISVALIDREF_statOff) THEN
  	IF (StrDs.ISVALIDREF_statOn) AND (StrDs.ISVALIDREF_statOff) THEN
  	StrDs.reliability:= statOn_reliability AND statOff_reliability;
  		_statOn  := statOn;
  		_statOff := statOff;
  	ELSIF (StrDs.ISVALIDREF_statOn) THEN
                       StrDs.reliability:= statOn_reliability;
  		_statOn  := statOn;
  		_statOff := NOT statOn;
  	ELSIF (StrDs.ISVALIDREF_statOff) THEN
  		 StrDs.reliability:= statOff_reliability;
  		_statOn  := NOT statOff;
  		_statOff :=statOff;
  	END_IF;

  	IF StrDs.reliability THEN
  		IF _statOn AND NOT _statOff 		THEN 	StrDs.onStatus := _statusDualInput.STATUS_ON;
  		ELSIF _statOff AND NOT _statOn 	THEN 	StrDs.onStatus := _statusDualInput.Status_OFF;
  		ELSIF NOT _statOn AND NOT _statOff 	THEN 	StrDs.onStatus := _statusDualInput.STATUS_TRANSITIONAL;
  		ELSE					StrDs.onStatus := _statusDualInput.STATUS_ERROR;
                      END_IF;

  	ELSE
  		StrDs.onStatus := _statusDualInput.STATUS_NOTDEFINED;

  	END_IF;
  ELSE
  	CASE BYTE_TO_INT(lastCmd) OF
  		(*baseCmdOn*) 1: StrDs.onStatus  := _statusDualInput.STATUS_ON;
  		(*baseCmdOff*) 2: StrDs.onStatus  := _statusDualInput.STATUS_OFF;

  	ELSE
  		 StrDs.onStatus := _statusDualInput.STATUS_NOTDEFINED;

  	END_CASE;
  END_IF;

  (* ---- Формирование признака сдвига ---- *)
  getSdvig := FALSE;
  IF (StrDs.ISVALIDREF_cmdOn OR StrDs.ISVALIDREF_cmdOff) THEN
  	IF NOT (StrDs.CmdOn OR StrDs.CmdOff) THEN
                       IF (lastOnStatus <> StrDs.onStatus AND
  		(StrDs.onStatus <> _statusDualInput.STATUS_NOTDEFINED AND
                       StrDs.onStatus <> _statusDualInput.STATUS_ERROR)     AND
  		(lastOnStatus <> _statusDualInput.STATUS_NOTDEFINED   AND
                       lastOnStatus <> _statusDualInput.STATUS_ERROR))
                      THEN
  			getSdvig   := TRUE;
  		END_IF;
  	END_IF;
  END_IF;

  IF getSdvig THEN StrDs.sdvig:= TRUE; END_IF;

  sdvigReset(IN:=StrDs.sdvig, PT:=T#15S);

  IF sdvigReset.Q THEN StrDs.sdvig:=FALSE; END_IF;

  lastOnStatus := StrDs.onStatus;

  StrDs.Accident := inAccident.value AND inAccident.reliability;
  StrDs.Ns := inNs.value AND inNs.reliability;
  StrDs.OpcCommandsDisabled := StrDs.inOpcCommandsDisabled;

  (* ---- Распаковка команды ---- *)
  _sunpackerCommand(command := StrDs.inCommand);
  	cmd := _sunpackerCommand.cmd;
  	source := _sunpackerCommand.source;

  (* ---- Обработка команды ---- *)
  IF cmd <> 0 AND lastCmd <> cmd and (((NOT StrDs.opcCommandsDisabled) AND source > 0) OR source = 0) then
  	CASE BYTE_TO_INT(cmd) OF
  	(*cmd_open*) 1 :
  			IF  StrDs.ISVALIDREF_cmdOn THEN StrDs.CmdOn := TRUE;
  				IF StrDs.ISVALIDREF_cmdOff THEN StrDs.CmdOff := FALSE; END_IF;
  			ELSIF  StrDs.ISVALIDREF_cmdOff THEN StrDs.CmdOff := FALSE;  END_IF;
  			errorCMDTimer(IN := false);
  			_commandErrorTimer := true;
  			StrDs.lastCmdIsOn := true;
  	(*cmd_close*) 2 :
  			IF StrDs.ISVALIDREF_cmdOff THEN StrDs.CmdOff := TRUE;
  				IF StrDs.ISVALIDREF_cmdOn THEN StrDs.CmdOn := FALSE; END_IF;
  			ELSIF StrDs.ISVALIDREF_cmdOn THEN StrDs.CmdOn := FALSE; END_IF;
  			errorCMDTimer(IN := false);
  			_commandErrorTimer := true;
  			StrDs.lastCmdIsOn := false;
  	(*cmd_reset*) 3 :    IF StrDs.ISVALIDREF_statOn OR StrDs.ISVALIDREF_statOff THEN
  			StrDs.CmdOn := FALSE;
  			StrDs.CmdOff := FALSE;
                                lastCmd :=0;
  			_commandErrorTimer := false;
  			StrDs.lastCmdIsOn := false;
                                END_IF;
  	END_CASE;
  	source_for_Status := source;
  	cmd_for_Status := cmd;
  	command_error_for_Status := 0;
  END_IF;

  lastCmd := cmd;
  errorCMDTimer(In := _commandErrorTimer, PT :=T#10s);

  (* ---- алгоритм  для команды ВКЛючить ---- *)
  IF (StrDs.onStatus = _statusDualInput.STATUS_ON) and (lastCmd = _commandDualInput.CMD_ON) then
  	IF StrDs.ISVALIDREF_cmdOn AND StrDs.ISVALIDREF_cmdOff then  StrDs.cmdOn := false; END_IF;

  	 errorCMDTimer(In := false);
  	 _commandErrorTimer := false;
  	 cmd_for_Status := 0;
  	 source_for_Status := 0;
  END_IF;

  (* ---- off ---- *)
  IF (StrDs.onStatus = _statusDualInput.STATUS_OFF) and (lastCmd = _commandDualInput.CMD_OFF) then
  	IF StrDs.ISVALIDREF_cmdOn AND StrDs.ISVALIDREF_cmdOff then  StrDs.cmdOff := false; END_IF;

  	 errorCMDTimer(In := false);
  	 _commandErrorTimer := false;
  	 cmd_for_Status := 0;
  	 source_for_Status := 0;
  END_IF;

  (* ---- ошибка исполнения команды ---- *)
  if errorCMDTimer.Q and (cmd_for_Status <> 0) then
  	command_error_for_Status :=  cmd_for_Status;
  	_commandErrorTimer := false;
  	StrDs.CmdOn := false;
  	StrDs.CmdOff := false;
  	lastCmd := 0;
  end_if;

  (* ---- сброс ошибки команды ---- *)
  StrDs.CommandFault := command_error_for_Status <> 0;
  _errorReset(IN := command_error_for_Status <> 0, PT := T#15S);
  IF _errorReset.Q THEN
  	cmd_for_Status := 0;
  	source_for_Status := 0;
  	command_error_for_Status := 0;
  END_IF;

  cmdOn := StrDs.cmdOn;
  cmdOff:= StrDs.cmdOff;

  (* ---- формирование зашифрованного статуса для АРМа ---- *)
  StrDs.status := shl(BYTE_TO_DWORD(source_for_Status), 29)
  		OR shl(BYTE_TO_DWORD(cmd_for_Status), 26)
  		OR shl(BYTE_TO_DWORD(command_error_for_Status), 23)
  		OR shl(bool_to_DWORD(StrDs.sdvig), 22)
  		OR shl(bool_to_DWORD(StrDs.OpcCommandsDisabled), 21)
  		OR shl(BOOL_TO_DWORD(StrDs.Ns), 4)
                  	OR shl(BOOL_TO_DWORD(StrDs.Accident ),3)
  		OR BYTE_TO_DWORD(StrDs.onStatus);
END_FUNCTION_BLOCK

FUNCTION_BLOCK fb_DO_Init
  VAR_INPUT
    data_Ini : BOOL;
    imit : BOOL      := FALSE;
  END_VAR
  VAR_IN_OUT
    strDO : struct_DO;
  END_VAR
  VAR_OUTPUT
    Init : BOOL      := FALSE;
  END_VAR

  (*****            Функциональный блок переинициализации структуры-дескриптора канала дискретного ввода.            *****)
   Init := FALSE;

      IF data_Ini THEN                            (* Параметрам требуется переинициализация. *)
          strDO.imit       := imit;
          data_Ini:=FALSE;
          Init := TRUE;
      END_IF;
    IF Init THEN
  imit:=FALSE;
     END_IF;
END_FUNCTION_BLOCK

FUNCTION_BLOCK fb_AiProtection
  VAR_INPUT
    ai : struct_AI;
  END_VAR
  VAR_IN_OUT
    StrAIp : struct_AiProtection;
  END_VAR
  VAR
    _sunpackerCommand : fb_sunpackerCommand;
    _signalingTp : TOF;
    _statusAi : TYPE_StatusAi;
    source : BYTE;
    cmd : BYTE;
    lastCmd : BYTE;
    source_for_Status : BYTE;
    cmd_for_Status : BYTE;
    command_error_for_Status : BYTE;
    resetCmdTimer : TON;
    resetCmdTimerPriznak : BOOL;
    signalinTimer : TON;
    timer : TON;
    SignalingTrig : R_TRIG;
    SignalingFTrig : F_TRIG;
    SignalingAi : BOOL;
  END_VAR

  timer(IN :=(ai.interval=StrAIp.controlLimit) AND (ai.interval >= _statusAi.normal) AND StrAIp.isRunning, PT :=StrAIp.delay);
  SignalingTrig(CLK := timer.Q);
  IF SignalingTrig.Q THEN
  	SignalingAi := TRUE;
  END_IF;
  SignalingFTrig(CLK := timer.Q);
  IF SignalingFTrig.Q THEN
  	SignalingAi := FALSE;
  END_IF;

  StrAIp.Tag := StrAIp.inTag;
  StrAIp.RunOnStart := StrAIp.inRunOnStart;

  StrAIp.CanRun := StrAIp.inCanRun;

  StrAIp.OpcCommandsDisabled := StrAIp.inOpcCommandsDisabled;

  (* ---- Если управление с ВУ заблокировано, то передаем команду из алгоритма ---- *)
  IF StrAIp.inOpcCommandsDisabled THEN
  	StrAIp.inCommand := StrAIp.inCommand_Alg;
  ELSE (* иначе передаем команду с АРМа*)
  	StrAIp.inCommand := StrAIp.inCommand_ARM;
  END_IF;

  _sunpackerCommand(command := StrAIp.inCommand);
  	source := _sunpackerCommand.source;
  	cmd := _sunpackerCommand.cmd;

  IF cmd <> 0 AND lastCmd <> cmd AND (((NOT StrAIp.opcCommandsDisabled) AND source > 0) OR source = 0) then

  	CASE BYTE_TO_INT(cmd) OF
  		(*cmdRun*) 1: 	IF        NOT StrAIp.Remont THEN
  					StrAIp.isEnded := FALSE;
  					StrAIp.hasError 	:= FALSE;
  					StrAIp.isRunning := TRUE;

  					cmd_for_Status := cmd;
  					source_for_Status := source;
  					command_error_for_Status := 0;
  				ELSE
  					StrAIp.isRunning := FALSE;
  					StrAIp.isEnded := FALSE;
  					StrAIp.hasError 	:= FALSE;

  					cmd_for_Status := 0;
  					source_for_Status := source;
  					command_error_for_Status := cmd;
  				END_IF;
                                          StrAIp.inopcCommandsDisabled:=FALSE;

  		(*cmdReset*) 2: 	StrAIp.isRunning := FALSE;
  				StrAIp.isEnded := FALSE;
  				StrAIp.hasError 	:= FALSE;
  				SignalingAi := FALSE;
  				StrAIp.Check := FALSE;
                                          (*StrAIp.Remont := FALSE;*)
  				cmd_for_Status := cmd;
  				source_for_Status := source;
  				command_error_for_Status := 0;
                                          StrAIp.inopcCommandsDisabled:=FALSE;

  	(*cmd_setRemont*) 4 :	StrAIp.Remont := TRUE;
  				(*StrAIp.isRunning := FALSE;*)

  				cmd_for_Status := cmd;
  				source_for_Status := source;
  				command_error_for_Status := 0;
  	(*cmd_resetRemont*) 5 : 	(*IF (ai.interval=StrAIp.controlLimit) THEN
  					cmd_for_Status := 0;
  					source_for_Status := 0;
  					command_error_for_Status := cmd;
  				ELSE*)
  					StrAIp.Remont := FALSE;
  					(*StrAIp.isRunning := TRUE;*)

  					cmd_for_Status := cmd;
  					source_for_Status := source;
  					command_error_for_Status := 0;
  				(*END_IF;*)
  	(*cmd_setCheck*) 6 : 	StrAIp.Check := TRUE;

  				cmd_for_Status := cmd;
  				source_for_Status := source;
  				command_error_for_Status := 0;
  	END_CASE;
  	resetCmdTimer(IN := false);
  	resetCmdTimerPriznak := TRUE;
  END_IF;
  lastCmd := cmd;

  resetCmdTimer(IN := resetCmdTimerPriznak);
  IF resetCmdTimer.Q THEN
  	resetCmdTimerPriznak := FALSE;
  	source_for_Status := 0;
  	cmd_for_Status := 0;
  	command_error_for_Status := 0;
  END_IF;

  IF StrAIp.isRunning AND NOT StrAIp.Remont AND NOT StrAIp.Check THEN
  	StrAIp.Signaling := SignalingAi;
  	StrAIp.SignalingTP := _signalingTp.Q;
  ELSE
  	StrAIp.Signaling := 0;
  	StrAIp.SignalingTP := 0;
  END_IF;

  _signalingTp(in := StrAIp.Signaling, PT := T#1s);

  StrAIp.status :=  SHL(BYTE_TO_DWORD(source_for_Status), 29)
  			OR SHL(BYTE_TO_DWORD(cmd_for_Status), 26)
  			OR SHL(BYTE_TO_DWORD(command_error_for_Status), 23)
  			OR SHL(BOOL_TO_DWORD(StrAIp.OpcCommandsDisabled ), 21)
  			OR SHL(BOOL_TO_DWORD(StrAIp.Signaling), 16)
  			OR SHL(BOOL_TO_DWORD(StrAIp.RunOnStart ), 15)
  			OR SHL(BOOL_TO_DWORD(StrAIp.remont), 6)
  			OR SHL(BOOL_TO_DWORD(StrAIp.Check), 5)
  			OR SHL(BOOL_TO_DWORD(StrAIp.hasError), 4)
  			OR SHL(BOOL_TO_DWORD(StrAIp.SignalingTP), 3)
  			OR SHL(BOOL_TO_DWORD(StrAIp.CanRun), 2)
  			OR SHL(BOOL_TO_DWORD(StrAIp.isEnded), 1)
  			OR BOOL_TO_DWORD(StrAIp.isRunning);
END_FUNCTION_BLOCK

FUNCTION_BLOCK ExtNarabotka
  VAR
    saveInterval : TIME      := T#30S;
    narabotka : UDINT;
    timer : RTC;
    saveTimer : TON;
  END_VAR
  VAR_IN_OUT
    retain_narabotka : UDINT;
  END_VAR
  VAR
    initialized : BOOL;
  END_VAR
  VAR_INPUT
    started : BOOL;
    reset : BOOL;
  END_VAR

  IF NOT initialized THEN
  	narabotka:=retain_narabotka;
  	initialized:=TRUE;
  END_IF;

  timer();

  IF timer.Q THEN
  	narabotka:=DT_TO_UDINT( timer.CDT);

  END_IF;
  saveTimer(IN:=TRUE, PT:=saveInterval);
  IF saveTimer.Q THEN
  	retain_narabotka:=narabotka;
  	saveTimer(IN:=FALSE);
  END_IF;

  IF started THEN
  	IF NOT timer.Q THEN
  		timer.PDT:=UDINT_TO_DT(narabotka);
                      timer.IN:=TRUE;
  	END_IF;
  ELSE
  	IF timer.Q THEN
  		timer.IN:=FALSE;
                      saveTimer.IN:=FALSE;
  	END_IF;
  END_IF;

  IF reset THEN
  timer.PDT:=UINT_TO_DT(0);
  IF timer.IN THEN
  	timer(IN:=FALSE);
  	timer(IN:=TRUE);
  END_IF;
  narabotka:=0;
  reset:=FALSE;
  END_IF;
END_FUNCTION_BLOCK

FUNCTION runIfNotRunningSO : BOOL
  VAR_IN_OUT
    so : struct_singleOutput;
  END_VAR
  VAR CONSTANT
    cmdRun : WORD      := 1;
  END_VAR

  IF NOT so.Q THEN
                      so.inOpcCommandsDisabled:=TRUE;
  		so.inCommand_Alg:=cmdRun;
  END_IF;
END_FUNCTION

FUNCTION resetIfRunningSO : BOOL
  VAR_IN_OUT
    so : struct_singleOutput;
  END_VAR
  VAR CONSTANT
    cmdReset : WORD      := 2;
  END_VAR

  IF so.Q THEN
                      so.inOpcCommandsDisabled:=TRUE;
  		so.inCommand_Alg:=cmdReset;
  END_IF;
END_FUNCTION

FUNCTION_BLOCK ph_SingleOutput
  VAR_IN_OUT
    im : struct_singleOutput;
  END_VAR
  VAR_INPUT
    WhatCanIdo : BOOL;
    PhaseNumber : UINT;
  END_VAR
  VAR_IN_OUT
    StrPh : struct_PhaseAlgoritm;
  END_VAR
  VAR
    reset_Trig : R_TRIG;
  END_VAR

  IF StrPh.run AND NOT StrPh.start THEN
  	StrPh.start := TRUE;
  	StrPh.top := FALSE;
  	StrPh.error := FALSE;
            StrPh.run:=FALSE;

  	IF (WhatCanIdo) THEN
  	runIfNotRunningSO(im);
            ELSE
  	resetIfRunningSO(im);
            END_IF;
  END_IF;

  IF StrPh.start AND NOT StrPh.top THEN
  StrPh.top := (im.Q = WhatCanIdo);
  END_IF;

  reset_Trig(CLK := StrPh.reset);
  IF reset_Trig.Q THEN
  	StrPh.start := FALSE;
  	StrPh.error := FALSE;
  	StrPh.top := FALSE;
            StrPh.run:=FALSE;
            StrPh.reset:=FALSE;
  END_IF;

  StrPh.startStatus := SHL(BOOL_TO_DWORD(StrPh.start), PhaseNumber);
  StrPh.errorStatus := SHL(BOOL_TO_DWORD(StrPh.error), PhaseNumber);
  StrPh.topStatus := SHL(BOOL_TO_DWORD(StrPh.top), PhaseNumber);
END_FUNCTION_BLOCK

FUNCTION_BLOCK OPC_PROTECTIONS_SET
  VAR_EXTERNAL
    protections_Topornogo_podshipnika_EDT_1_status : UDINT;
    protections_Toy_podshipnika_EDT_2_status : UDINT;
    protections_Toy_podshipnika_kol_EDT_3_status : UDINT;
    protections_Toy_podshipnika_kol_EDT_4_status : UDINT;
    protections_To_podshipnika_shest_red_EDT_5_status : UDINT;
    protections_To_podshipnika_shest_red_EDT_6_status : UDINT;
    protections_To_podshipnika_N_EDT_7_status : UDINT;
    protections_To_podshipnika_svob_konca_EDT_8_status : UDINT;
    protections_Ty_podshipnika_rab_kol_EDT_9_status : UDINT;
    protections_Typornogo_podshipnika_nerab_kolodok_HT_10_status : UDINT;
    protections_Tgaza_na_vyhode_H_status : UDINT;
    protections_Os_sdvig_nagnetatelja_plus_status : UDINT;
    protections_Os_sdvig_nagnetatelja_minus_status : UDINT;
    protections_Pgaza_na_vyhode_nagnetatelia_GPA_STOP_status : UDINT;
    protections_Pgaza_na_vhode_nagnetatelia_GPA_STOP_status : UDINT;
    protections_Pgaza_na_vyhode_nagnetatelia_status : UDINT;
    protections_dPmaslo_gaz_status : UDINT;
    protections_Pmaslo_sm_nizkoe_status : UDINT;
    protections_Pmaslo_sm_vysokoe_status : UDINT;
    protections_Vibro_skorost_OPED_T1_status : UDINT;
    protections_Vibro_skorost_OPED_T2_status : UDINT;
    protections_Vibro_skorost_OYP_kolesa_ED_T3_status : UDINT;
    protections_Vibro_skorost_OP_kolesa_RH_T4_status : UDINT;
    protections_Vibro_skorost_OP_shesterni_RED_T5_status : UDINT;
    protections_Vibro_skorost_OP_shesterni_RED_T6_status : UDINT;
    protections_dPmaslo_gaz_less100_status : UDINT;
    protections_Reg_vozb_off_status : UDINT;
    protections_Fprotectionsl_chastotnii_pusk_status : UDINT;
    protections_Off_avar_vikluchatel_status : UDINT;
    protections_AOKC_SHKC_status : UDINT;
    protections_AO_PRU_status : UDINT;
    protections_AO_ot_SHU_status : UDINT;
    protections_mvOff_status : UDINT;
    protections_Kran1_sdvig_status : UDINT;
    protections_Kran2_sdvig_status : UDINT;
  END_VAR

  protections_Topornogo_podshipnika_EDT_1_status := DWORD_TO_UDINT(protections.Topornogo_podshipnika_EDT_1.status);

  protections_Toy_podshipnika_EDT_2_status := DWORD_TO_UDINT(protections.Toy_podshipnika_EDT_2.status);

  protections_Toy_podshipnika_kol_EDT_3_status := DWORD_TO_UDINT(protections.Toy_podshipnika_kol_EDT_3.status);

  protections_Toy_podshipnika_kol_EDT_4_status := DWORD_TO_UDINT(protections.Toy_podshipnika_kol_EDT_4.status);

  protections_To_podshipnika_shest_red_EDT_5_status := DWORD_TO_UDINT(protections.To_podshipnika_shest_red_EDT_5.status);

  protections_To_podshipnika_shest_red_EDT_6_status := DWORD_TO_UDINT(protections.To_podshipnika_shest_red_EDT_6.status);

  protections_To_podshipnika_N_EDT_7_status := DWORD_TO_UDINT(protections.To_podshipnika_N_EDT_7.status);

  protections_To_podshipnika_svob_konca_EDT_8_status := DWORD_TO_UDINT(protections.To_podshipnika_svob_konca_EDT_8.status);

  protections_Ty_podshipnika_rab_kol_EDT_9_status := DWORD_TO_UDINT(protections.Ty_podshipnika_rab_kol_EDT_9.status);

  protections_Typornogo_podshipnika_nerab_kolodok_HT_10_status := DWORD_TO_UDINT(protections.Typornogo_podshipnika_nerab_kolodok_HT_10.status);

  protections_Tgaza_na_vyhode_H_status := DWORD_TO_UDINT(protections.Tgaza_na_vyhode_H.status);

  protections_Os_sdvig_nagnetatelja_plus_status := DWORD_TO_UDINT(protections.Os_sdvig_nagnetatelja_plus.status);

  protections_Os_sdvig_nagnetatelja_minus_status := DWORD_TO_UDINT(protections.Os_sdvig_nagnetatelja_minus.status);

  protections_Pgaza_na_vyhode_nagnetatelia_GPA_STOP_status := DWORD_TO_UDINT(protections.Pgaza_na_vyhode_nagnetatelia_GPA_STOP.status);

  protections_Pgaza_na_vhode_nagnetatelia_GPA_STOP_status := DWORD_TO_UDINT(protections.Pgaza_na_vhode_nagnetatelia_GPA_STOP.status);

  protections_Pgaza_na_vyhode_nagnetatelia_status := DWORD_TO_UDINT(protections.Pgaza_na_vyhode_nagnetatelia.status);

  protections_dPmaslo_gaz_status := DWORD_TO_UDINT(protections.dPmaslo_gaz.status);

  protections_Pmaslo_sm_nizkoe_status := DWORD_TO_UDINT(protections.Pmaslo_sm_nizkoe.status);

  protections_Pmaslo_sm_vysokoe_status := DWORD_TO_UDINT(protections.Pmaslo_sm_vysokoe.status);

  protections_Vibro_skorost_OPED_T1_status := DWORD_TO_UDINT(protections.Vibro_skorost_OPED_T1.status);

  protections_Vibro_skorost_OPED_T2_status := DWORD_TO_UDINT(protections.Vibro_skorost_OPED_T2.status);

  protections_Vibro_skorost_OYP_kolesa_ED_T3_status := DWORD_TO_UDINT(protections.Vibro_skorost_OYP_kolesa_ED_T3.status);

  protections_Vibro_skorost_OP_kolesa_RH_T4_status := DWORD_TO_UDINT(protections.Vibro_skorost_OP_kolesa_RH_T4.status);

  protections_Vibro_skorost_OP_shesterni_RED_T5_status := DWORD_TO_UDINT(protections.Vibro_skorost_OP_shesterni_RED_T5.status);

  protections_Vibro_skorost_OP_shesterni_RED_T6_status := DWORD_TO_UDINT(protections.Vibro_skorost_OP_shesterni_RED_T6.status);

  protections_dPmaslo_gaz_less100_status := DWORD_TO_UDINT(protections.dPmaslo_gaz_less100.status);

  protections_Reg_vozb_off_status := DWORD_TO_UDINT(protections.Reg_vozb_off.status);

  protections_Fprotectionsl_chastotnii_pusk_status := DWORD_TO_UDINT(protections.Fprotectionsl_chastotnii_pusk.status);

  protections_Off_avar_vikluchatel_status := DWORD_TO_UDINT(protections.Off_avar_vikluchatel.status);

  protections_AOKC_SHKC_status := DWORD_TO_UDINT(protections.AOKC_SHKC.status);

  protections_AO_PRU_status := DWORD_TO_UDINT(protections.AO_PRU.status);

  protections_AO_ot_SHU_status := DWORD_TO_UDINT(protections.AO_ot_SHU.status);

  protections_mvOff_status := DWORD_TO_UDINT(protections.mvOff.status);

  protections_Kran1_sdvig_status := DWORD_TO_UDINT(protections.Kran1_sdvig.status);

  protections_Kran2_sdvig_status := DWORD_TO_UDINT(protections.Kran2_sdvig.status);
END_FUNCTION_BLOCK

FUNCTION_BLOCK OPC_PROTECTIONS_GET
  VAR_EXTERNAL
    protections_Topornogo_podshipnika_EDT_1_command : UINT;
    protections_Toy_podshipnika_EDT_2_command : UINT;
    protections_Toy_podshipnika_kol_EDT_3_command : UINT;
    protections_Toy_podshipnika_kol_EDT_4_command : UINT;
    protections_To_podshipnika_shest_red_EDT_5_command : UINT;
    protections_To_podshipnika_shest_red_EDT_6_command : UINT;
    protections_To_podshipnika_N_EDT_7_command : UINT;
    protections_To_podshipnika_svob_konca_EDT_8_command : UINT;
    protections_Ty_podshipnika_rab_kol_EDT_9_command : UINT;
    protections_Typornogo_podshipnika_nerab_kolodok_HT_10_command : UINT;
    protections_Tgaza_na_vyhode_H_command : UINT;
    protections_Os_sdvig_nagnetatelja_plus_command : UINT;
    protections_Os_sdvig_nagnetatelja_minus_command : UINT;
    protections_Pgaza_na_vyhode_nagnetatelia_GPA_STOP_command : UINT;
    protections_Pgaza_na_vhode_nagnetatelia_GPA_STOP_command : UINT;
    protections_Pgaza_na_vyhode_nagnetatelia_command : UINT;
    protections_dPmaslo_gaz_command : UINT;
    protections_Pmaslo_sm_nizkoe_command : UINT;
    protections_Pmaslo_sm_vysokoe_command : UINT;
    protections_Vibro_skorost_OPED_T1_command : UINT;
    protections_Vibro_skorost_OPED_T2_command : UINT;
    protections_Vibro_skorost_OYP_kolesa_ED_T3_command : UINT;
    protections_Vibro_skorost_OP_kolesa_RH_T4_command : UINT;
    protections_Vibro_skorost_OP_shesterni_RED_T5_command : UINT;
    protections_Vibro_skorost_OP_shesterni_RED_T6_command : UINT;
    protections_dPmaslo_gaz_less100_command : UINT;
    protections_Reg_vozb_off_command : UINT;
    protections_Fprotectionsl_chastotnii_pusk_command : UINT;
    protections_Off_avar_vikluchatel_command : UINT;
    protections_AOKC_SHKC_command : UINT;
    protections_AO_PRU_command : UINT;
    protections_AO_ot_SHU_command : UINT;
    protections_mvOff_command : UINT;
    protections_Kran1_sdvig_command : UINT;
    protections_Kran2_sdvig_command : UINT;
  END_VAR

  protections.Topornogo_podshipnika_EDT_1.inCommand_ARM := UINT_TO_WORD(protections_Topornogo_podshipnika_EDT_1_command);

  protections.Toy_podshipnika_EDT_2.inCommand_ARM := UINT_TO_WORD(protections_Toy_podshipnika_EDT_2_command);

  protections.Toy_podshipnika_kol_EDT_3.inCommand_ARM := UINT_TO_WORD(protections_Toy_podshipnika_kol_EDT_3_command);

  protections.Toy_podshipnika_kol_EDT_4.inCommand_ARM := UINT_TO_WORD(protections_Toy_podshipnika_kol_EDT_4_command);

  protections.To_podshipnika_shest_red_EDT_5.inCommand_ARM := UINT_TO_WORD(protections_To_podshipnika_shest_red_EDT_5_command);

  protections.To_podshipnika_shest_red_EDT_6.inCommand_ARM := UINT_TO_WORD(protections_To_podshipnika_shest_red_EDT_6_command);

  protections.To_podshipnika_N_EDT_7.inCommand_ARM := UINT_TO_WORD(protections_To_podshipnika_N_EDT_7_command);

  protections.To_podshipnika_svob_konca_EDT_8.inCommand_ARM := UINT_TO_WORD(protections_To_podshipnika_svob_konca_EDT_8_command);

  protections.Ty_podshipnika_rab_kol_EDT_9.inCommand_ARM := UINT_TO_WORD(protections_Ty_podshipnika_rab_kol_EDT_9_command);

  protections.Typornogo_podshipnika_nerab_kolodok_HT_10.inCommand_ARM := UINT_TO_WORD(protections_Typornogo_podshipnika_nerab_kolodok_HT_10_command);

  protections.Tgaza_na_vyhode_H.inCommand_ARM := UINT_TO_WORD(protections_Tgaza_na_vyhode_H_command);

  protections.Os_sdvig_nagnetatelja_plus.inCommand_ARM := UINT_TO_WORD(protections_Os_sdvig_nagnetatelja_plus_command);

  protections.Os_sdvig_nagnetatelja_minus.inCommand_ARM := UINT_TO_WORD(protections_Os_sdvig_nagnetatelja_minus_command);

  protections.Pgaza_na_vyhode_nagnetatelia_GPA_STOP.inCommand_ARM := UINT_TO_WORD(protections_Pgaza_na_vyhode_nagnetatelia_GPA_STOP_command);

  protections.Pgaza_na_vhode_nagnetatelia_GPA_STOP.inCommand_ARM := UINT_TO_WORD(protections_Pgaza_na_vhode_nagnetatelia_GPA_STOP_command);

  protections.Pgaza_na_vyhode_nagnetatelia.inCommand_ARM := UINT_TO_WORD(protections_Pgaza_na_vyhode_nagnetatelia_command);

  protections.dPmaslo_gaz.inCommand_ARM := UINT_TO_WORD(protections_dPmaslo_gaz_command);

  protections.Pmaslo_sm_nizkoe.inCommand_ARM := UINT_TO_WORD(protections_Pmaslo_sm_nizkoe_command);

  protections.Pmaslo_sm_vysokoe.inCommand_ARM := UINT_TO_WORD(protections_Pmaslo_sm_vysokoe_command);

  protections.Vibro_skorost_OPED_T1.inCommand_ARM := UINT_TO_WORD(protections_Vibro_skorost_OPED_T1_command);

  protections.Vibro_skorost_OPED_T2.inCommand_ARM := UINT_TO_WORD(protections_Vibro_skorost_OPED_T2_command);

  protections.Vibro_skorost_OYP_kolesa_ED_T3.inCommand_ARM := UINT_TO_WORD(protections_Vibro_skorost_OYP_kolesa_ED_T3_command);

  protections.Vibro_skorost_OP_kolesa_RH_T4.inCommand_ARM := UINT_TO_WORD(protections_Vibro_skorost_OP_kolesa_RH_T4_command);

  protections.Vibro_skorost_OP_shesterni_RED_T5.inCommand_ARM := UINT_TO_WORD(protections_Vibro_skorost_OP_shesterni_RED_T5_command);

  protections.Vibro_skorost_OP_shesterni_RED_T6.inCommand_ARM := UINT_TO_WORD(protections_Vibro_skorost_OP_shesterni_RED_T6_command);

  protections.dPmaslo_gaz_less100.inCommand_ARM := UINT_TO_WORD(protections_dPmaslo_gaz_less100_command);

  protections.Reg_vozb_off.inCommand_ARM := UINT_TO_WORD(protections_Reg_vozb_off_command);

  protections.Fprotectionsl_chastotnii_pusk.inCommand_ARM := UINT_TO_WORD(protections_Fprotectionsl_chastotnii_pusk_command);

  protections.Off_avar_vikluchatel.inCommand_ARM := UINT_TO_WORD(protections_Off_avar_vikluchatel_command);

  protections.AOKC_SHKC.inCommand_ARM := UINT_TO_WORD(protections_AOKC_SHKC_command);

  protections.AO_PRU.inCommand_ARM := UINT_TO_WORD(protections_AO_PRU_command);

  protections.AO_ot_SHU.inCommand_ARM := UINT_TO_WORD(protections_AO_ot_SHU_command);

  protections.mvOff.inCommand_ARM := UINT_TO_WORD(protections_mvOff_command);

  protections.Kran1_sdvig.inCommand_ARM := UINT_TO_WORD(protections_Kran1_sdvig_command);

  protections.Kran2_sdvig.inCommand_ARM := UINT_TO_WORD(protections_Kran2_sdvig_command);
END_FUNCTION_BLOCK

FUNCTION_BLOCK OPC_IM_SET
  VAR_EXTERNAL
    IM_Kran1_status : UDINT;
    IM_Kran2_status : UDINT;
    IM_Kran3_status : UDINT;
    IM_Kran3b_status : UDINT;
    IM_Kran4_status : UDINT;
    IM_Kran5_status : UDINT;
    IM_Kran6_status : UDINT;
    IM_nu1_status : UDINT;
    IM_nu2_status : UDINT;
    IM_pns_status : UDINT;
    IM_v1_Avom_status : UDINT;
    IM_v2_Avom_status : UDINT;
    IM_v3_Avom_status : UDINT;
    IM_v4_Avom_status : UDINT;
    IM_mv_status : UDINT;
    IM_Reserve_IM1_status : UDINT;
    IM_Reserve_IM2_status : UDINT;
    IM_SingleSignals_status : UDINT;
    IM_SingleOutputs_status : UDINT;
    IM_KaloriferAVOM_status : UDINT;
    IM_CMN_status : UDINT;
    IM_TEN_kollectora_status : UDINT;
    IM_TEN_MB_status : UDINT;
    IM_SingleSignals_dP_maslo_gaz_Less100_status : UDINT;
    IM_SingleSignals_dp_kran1_Less100_status : UDINT;
    IM_SingleSignals_Razreshenie_zagruzki_dvig_status : UDINT;
    IM_SingleSignals_Vozbud_gotovnost_status : UDINT;
    IM_SingleSignals_Vozbud_neispr_tsepey_upr_AVR_pit_status : UDINT;
    IM_SingleSignals_Vozbud_neispravnost_status : UDINT;
    IM_SingleSignals_SHAVR1_v_rabote_status : UDINT;
    IM_SingleSignals_SHAVR2_v_rabote_status : UDINT;
    IM_SingleSignals_Avariinoe_otkluch_vikluchatelya_status : UDINT;
    IM_SingleSignals_Assinhronnii_hod_peregruzka_status : UDINT;
    IM_SingleSignals_SHU_v_GPA_vkluch_status : UDINT;
    IM_SingleSignals_SHP_v_GPA_vkluch_status : UDINT;
    IM_SingleSignals_QF1_on_status : UDINT;
    IM_SingleSignals_QF2_on_status : UDINT;
    IM_SingleSignals_QF23_on_status : UDINT;
    IM_SingleSignals_QF4_QF5_on_status : UDINT;
    IM_SingleSignals_QF6_QF7_on_status : UDINT;
    IM_SingleSignals_QF8_QF9_on_status : UDINT;
    IM_SingleSignals_QF10_QF11_on_status : UDINT;
    IM_SingleSignals_QF12_QF13_on_status : UDINT;
    IM_SingleSignals_QF14_QF15_on_status : UDINT;
    IM_SingleSignals_QF22_on_status : UDINT;
    IM_SingleSignals_NS_G1_G2_status : UDINT;
    IM_SingleSignals_NS_G3_G4_status : UDINT;
    IM_SingleSignals_NS_G15_G16_status : UDINT;
    IM_SingleSignals_NS_G17_status : UDINT;
    IM_SingleSignals_NS_G5_G6_status : UDINT;
    IM_SingleSignals_NS_G7_G8_status : UDINT;
    IM_SingleSignals_NS_G18_G19_status : UDINT;
    IM_SingleSignals_NS_G10_G11_status : UDINT;
    IM_SingleSignals_NS_G13_G14_status : UDINT;
    IM_SingleSignals_Uroven_masla_akkum_status : UDINT;
    IM_SingleSignals_NKU1_GPA_on_status : UDINT;
    IM_SingleSignals_NKU2_GPA_on_status : UDINT;
    IM_SingleSignals_AO_KC_ot_SHKS_status : UDINT;
    IM_SingleSignals_AO_GPA_ot_SHU_status : UDINT;
    IM_SingleSignals_BEAO_srabotal_status : UDINT;
    IM_SingleSignals_Chastotny_pusk_status : UDINT;
    IM_SingleSignals_Neuspesh_chastotny_pusk_status : UDINT;
    IM_SingleSignals_Rezhim_ruchnogo_regulirovaniya_status : UDINT;
    IM_SingleSignals_Osnovnoy_regul_off_status : UDINT;
    IM_SingleSignals_Voltage_sekcii_norm_status : UDINT;
    IM_SingleSignals_Reactorny_pusk_status : UDINT;
    IM_SingleSignals_NO_GPA_ot_SHU_status : UDINT;
    IM_SingleSignals_AO_GPA_ot_PRU_status : UDINT;
    IM_SingleSignals_Nalichie_BP1_status : UDINT;
    IM_SingleSignals_Nalichie_BP2_status : UDINT;
    IM_SingleSignals_Nalichie_BP3_status : UDINT;
    IM_SingleSignals_Nalichie_BP4_status : UDINT;
    IM_SingleSignals_Nalichie_BP5_status : UDINT;
    IM_SingleSignals_Nalichie_BP6_status : UDINT;
    IM_SingleSignals_Nalichie_BP7_BP8_status : UDINT;
    IM_SingleSignals_Nalichie_BP9_BP10_status : UDINT;
    IM_SingleSignals_Nalichie_cepei_upravlen_mv_status : UDINT;
    IM_SingleSignals_Nalichie_220BEAO_status : UDINT;
    IM_SingleSignals_Nalichie_per_220_na_vhode_status : UDINT;
    IM_SingleSignals_Nalichie_post_220_na_vhode_status : UDINT;
    IM_SingleSignals_Nalichie_BP11_status : UDINT;
    IM_SingleSignals_Nalichie_BP12_status : UDINT;
    IM_SingleSignals_Dver_SHU_pered_otkrita_status : UDINT;
    IM_SingleSignals_Dver_SHU_zad_otkrita_status : UDINT;
    IM_SingleSignals_EO_GPA_ot_knopki_SHU_status : UDINT;
    IM_SingleSignals_EO_EGPA_ot_PRY_status : UDINT;
    IM_SingleSignals_Synchroniz_rezhima_K1_status : UDINT;
    IM_SingleSignals_Potok_ms_posle_AVOM_status : UDINT;
  END_VAR

  IM_Kran1_status := DWORD_TO_UDINT(im.Kran1.status);

  IM_Kran2_status := DWORD_TO_UDINT(im.Kran2.status);

  IM_Kran3_status := DWORD_TO_UDINT(im.Kran3.status);

  IM_Kran3b_status := DWORD_TO_UDINT(im.Kran3b.status);

  IM_Kran4_status := DWORD_TO_UDINT(im.Kran4.status);

  IM_Kran5_status := DWORD_TO_UDINT(im.Kran5.status);

  IM_Kran6_status := DWORD_TO_UDINT(im.Kran6.status);

  IM_nu1_status := DWORD_TO_UDINT(im.nu1.status);

  IM_nu2_status := DWORD_TO_UDINT(im.nu2.status);

  IM_pns_status := DWORD_TO_UDINT(im.pns.status);

  IM_v1_Avom_status := DWORD_TO_UDINT(im.v1_Avom.status);

  IM_v2_Avom_status := DWORD_TO_UDINT(im.v2_Avom.status);

  IM_v3_Avom_status := DWORD_TO_UDINT(im.v3_Avom.status);

  IM_v4_Avom_status := DWORD_TO_UDINT(im.v4_Avom.status);

  IM_mv_status := DWORD_TO_UDINT(im.mv.status);

  IM_KaloriferAVOM_status := DWORD_TO_UDINT(im.KaloriferAVOM.status);

  IM_CMN_status := DWORD_TO_UDINT(im.CMN.status);

  IM_TEN_kollectora_status := DWORD_TO_UDINT(im.TEN_kollectora.status);

  IM_TEN_MB_status := DWORD_TO_UDINT(im.TEN_MB.status);

  IM_SingleSignals_dP_maslo_gaz_Less100_status := DWORD_TO_UDINT(im.SingleSignals._dP_maslo_gaz_Less100.status);

  IM_SingleSignals_dp_kran1_Less100_status := DWORD_TO_UDINT(im.SingleSignals._dp_kran1_Less100.status);

  IM_SingleSignals_Razreshenie_zagruzki_dvig_status := DWORD_TO_UDINT(im.SingleSignals._Razreshenie_zagruzki_dvig.status);

  IM_SingleSignals_Vozbud_gotovnost_status := DWORD_TO_UDINT(im.SingleSignals._Vozbud_gotovnost.status);

  IM_SingleSignals_Vozbud_neispr_tsepey_upr_AVR_pit_status := DWORD_TO_UDINT(im.SingleSignals._Vozbud_neispr_tsepey_upr_AVR_pit.status);

  IM_SingleSignals_Vozbud_neispravnost_status := DWORD_TO_UDINT(im.SingleSignals._Vozbud_neispravnost.status);

  IM_SingleSignals_SHAVR1_v_rabote_status := DWORD_TO_UDINT(im.SingleSignals._SHAVR1_v_rabote.status);

  IM_SingleSignals_SHAVR2_v_rabote_status := DWORD_TO_UDINT(im.SingleSignals._SHAVR2_v_rabote.status);

  IM_SingleSignals_Avariinoe_otkluch_vikluchatelya_status := DWORD_TO_UDINT(im.SingleSignals._Avariinoe_otkluch_vikluchatelya.status);

  IM_SingleSignals_Assinhronnii_hod_peregruzka_status := DWORD_TO_UDINT(im.SingleSignals._Assinhronnii_hod_peregruzka.status);

  IM_SingleSignals_SHU_v_GPA_vkluch_status := DWORD_TO_UDINT(im.SingleSignals._SHU_v_GPA_vkluch.status);

  IM_SingleSignals_SHP_v_GPA_vkluch_status := DWORD_TO_UDINT(im.SingleSignals._SHP_v_GPA_vkluch.status);

  IM_SingleSignals_QF1_on_status := DWORD_TO_UDINT(im.SingleSignals._QF1_on.status);

  IM_SingleSignals_QF2_on_status := DWORD_TO_UDINT(im.SingleSignals._QF2_on.status);

  IM_SingleSignals_QF23_on_status := DWORD_TO_UDINT(im.SingleSignals._QF23_on.status);

  IM_SingleSignals_QF4_QF5_on_status := DWORD_TO_UDINT(im.SingleSignals._QF4_QF5_on.status);

  IM_SingleSignals_QF6_QF7_on_status := DWORD_TO_UDINT(im.SingleSignals._QF6_QF7_on.status);

  IM_SingleSignals_QF8_QF9_on_status := DWORD_TO_UDINT(im.SingleSignals._QF8_QF9_on.status);

  IM_SingleSignals_QF10_QF11_on_status := DWORD_TO_UDINT(im.SingleSignals._QF10_QF11_on.status);

  IM_SingleSignals_QF12_QF13_on_status := DWORD_TO_UDINT(im.SingleSignals._QF12_QF13_on.status);

  IM_SingleSignals_QF14_QF15_on_status := DWORD_TO_UDINT(im.SingleSignals._QF14_QF15_on.status);

  IM_SingleSignals_QF22_on_status := DWORD_TO_UDINT(im.SingleSignals._QF22_on.status);

  IM_SingleSignals_NS_G1_G2_status := DWORD_TO_UDINT(im.SingleSignals._NS_G1_G2.status);

  IM_SingleSignals_NS_G3_G4_status := DWORD_TO_UDINT(im.SingleSignals._NS_G3_G4.status);

  IM_SingleSignals_NS_G15_G16_status := DWORD_TO_UDINT(im.SingleSignals._NS_G15_G16.status);

  IM_SingleSignals_NS_G17_status := DWORD_TO_UDINT(im.SingleSignals._NS_G17.status);

  IM_SingleSignals_NS_G5_G6_status := DWORD_TO_UDINT(im.SingleSignals._NS_G5_G6.status);

  IM_SingleSignals_NS_G7_G8_status := DWORD_TO_UDINT(im.SingleSignals._NS_G7_G8.status);

  IM_SingleSignals_NS_G18_G19_status := DWORD_TO_UDINT(im.SingleSignals._NS_G18_G19.status);

  IM_SingleSignals_NS_G10_G11_status := DWORD_TO_UDINT(im.SingleSignals._NS_G10_G11.status);

  IM_SingleSignals_NS_G13_G14_status := DWORD_TO_UDINT(im.SingleSignals._NS_G13_G14.status);

  IM_SingleSignals_Uroven_masla_akkum_status := DWORD_TO_UDINT(im.SingleSignals._Uroven_masla_akkum.status);

  IM_SingleSignals_NKU1_GPA_on_status := DWORD_TO_UDINT(im.SingleSignals._NKU1_GPA_on.status);

  IM_SingleSignals_NKU2_GPA_on_status := DWORD_TO_UDINT(im.SingleSignals._NKU2_GPA_on.status);

  IM_SingleSignals_AO_KC_ot_SHKS_status := DWORD_TO_UDINT(im.SingleSignals._AO_KC_ot_SHKS.status);

  IM_SingleSignals_AO_GPA_ot_SHU_status := DWORD_TO_UDINT(im.SingleSignals._AO_GPA_ot_SHU.status);

  IM_SingleSignals_BEAO_srabotal_status := DWORD_TO_UDINT(im.SingleSignals._BEAO_srabotal.status);

  IM_SingleSignals_Chastotny_pusk_status := DWORD_TO_UDINT(im.SingleSignals._Chastotny_pusk.status);

  IM_SingleSignals_Neuspesh_chastotny_pusk_status := DWORD_TO_UDINT(im.SingleSignals._Neuspesh_chastotny_pusk.status);

  IM_SingleSignals_Rezhim_ruchnogo_regulirovaniya_status := DWORD_TO_UDINT(im.SingleSignals._Rezhim_ruchnogo_regulirovaniya.status);

  IM_SingleSignals_Osnovnoy_regul_off_status := DWORD_TO_UDINT(im.SingleSignals._Osnovnoy_regul_off.status);

  IM_SingleSignals_Voltage_sekcii_norm_status := DWORD_TO_UDINT(im.SingleSignals._Voltage_sekcii_norm.status);

  IM_SingleSignals_Reactorny_pusk_status := DWORD_TO_UDINT(im.SingleSignals._Reactorny_pusk.status);

  IM_SingleSignals_NO_GPA_ot_SHU_status := DWORD_TO_UDINT(im.SingleSignals._NO_GPA_ot_SHU.status);

  IM_SingleSignals_AO_GPA_ot_PRU_status := DWORD_TO_UDINT(im.SingleSignals._AO_GPA_ot_PRU.status);

  IM_SingleSignals_Nalichie_BP1_status := DWORD_TO_UDINT(im.SingleSignals._Nalichie_BP1.status);

  IM_SingleSignals_Nalichie_BP2_status := DWORD_TO_UDINT(im.SingleSignals._Nalichie_BP2.status);

  IM_SingleSignals_Nalichie_BP3_status := DWORD_TO_UDINT(im.SingleSignals._Nalichie_BP3.status);

  IM_SingleSignals_Nalichie_BP4_status := DWORD_TO_UDINT(im.SingleSignals._Nalichie_BP4.status);

  IM_SingleSignals_Nalichie_BP5_status := DWORD_TO_UDINT(im.SingleSignals._Nalichie_BP5.status);

  IM_SingleSignals_Nalichie_BP6_status := DWORD_TO_UDINT(im.SingleSignals._Nalichie_BP6.status);

  IM_SingleSignals_Nalichie_BP7_BP8_status := DWORD_TO_UDINT(im.SingleSignals._Nalichie_BP7_BP8.status);

  IM_SingleSignals_Nalichie_BP9_BP10_status := DWORD_TO_UDINT(im.SingleSignals._Nalichie_BP9_BP10.status);

  IM_SingleSignals_Nalichie_cepei_upravlen_mv_status := DWORD_TO_UDINT(im.SingleSignals._Nalichie_cepei_upravlen_mv.status);

  IM_SingleSignals_Nalichie_220BEAO_status := DWORD_TO_UDINT(im.SingleSignals._Nalichie_220BEAO.status);

  IM_SingleSignals_Nalichie_per_220_na_vhode_status := DWORD_TO_UDINT(im.SingleSignals._Nalichie_per_220_na_vhode.status);

  IM_SingleSignals_Nalichie_post_220_na_vhode_status := DWORD_TO_UDINT(im.SingleSignals._Nalichie_post_220_na_vhode.status);

  IM_SingleSignals_Nalichie_BP11_status := DWORD_TO_UDINT(im.SingleSignals._Nalichie_BP11.status);

  IM_SingleSignals_Nalichie_BP12_status := DWORD_TO_UDINT(im.SingleSignals._Nalichie_BP12.status);

  IM_SingleSignals_Dver_SHU_pered_otkrita_status := DWORD_TO_UDINT(im.SingleSignals._Dver_SHU_pered_otkrita.status);

  IM_SingleSignals_Dver_SHU_zad_otkrita_status := DWORD_TO_UDINT(im.SingleSignals._Dver_SHU_zad_otkrita.status);

  IM_SingleSignals_EO_GPA_ot_knopki_SHU_status := DWORD_TO_UDINT(im.SingleSignals._EO_GPA_ot_knopki_SHU.status);

  IM_SingleSignals_EO_EGPA_ot_PRY_status := DWORD_TO_UDINT(im.SingleSignals._EO_EGPA_ot_PRY.status);

  IM_SingleSignals_Synchroniz_rezhima_K1_status := DWORD_TO_UDINT(im.SingleSignals._Synchroniz_rezhima_K1.status);

  IM_SingleSignals_Potok_ms_posle_AVOM_status := DWORD_TO_UDINT(im.SingleSignals._Potok_ms_posle_AVOM.status);
END_FUNCTION_BLOCK

FUNCTION_BLOCK fb_meandr
  VAR
    _output : BOOL;
  END_VAR
  VAR_INPUT
    period : TIME      := T#300MS;
  END_VAR
  VAR
    timer : TON;
    FALSE_val : BOOL      := FALSE;
    TRUE_val : BOOL      := TRUE;
  END_VAR
  VAR_IN_OUT
    output : BOOL;
  END_VAR

  timer(in:=NOT FALSE_val,PT:=period);

  IF timer.Q THEN
      _output:=_output XOR TRUE_val;
      timer(in:=FALSE);
  END_IF;

  output:=_output;
END_FUNCTION_BLOCK

FUNCTION_BLOCK fb_Kran_Init
  VAR_INPUT
    data_Ini : BOOL;
    ISVALIDREF_statOn : BOOL;
    ISVALIDREF_statOff : BOOL;
    ISVALIDREF_cmdOn : BOOL;
    ISVALIDREF_cmdOff : BOOL;
    ISVALIDREF_inSo : BOOL;
    ISVALIDREF_inSz : BOOL;
    ISVALIDREF_inDp : BOOL      := False;
    continueHoldCommand : TIME;
  END_VAR
  VAR_IN_OUT
    str_Kr : struct_Kran;
  END_VAR
  VAR_OUTPUT
    Init : BOOL      := FALSE;
  END_VAR

  (*****            Функциональный блок переинициализации структуры  Kran          *****)

          Init := False;

      IF data_Ini THEN                            (* Параметрам требуется переинициализация. *)
          str_Kr.ISVALIDREF_statOn                := ISVALIDREF_statOn;
          str_Kr.ISVALIDREF_statOff               := ISVALIDREF_statOff;
          str_Kr.ISVALIDREF_cmdOn                 := ISVALIDREF_cmdOn;
          str_Kr.ISVALIDREF_cmdOff                := ISVALIDREF_cmdOff;
          str_Kr.ISVALIDREF_inSo                  := ISVALIDREF_inSo;
          str_Kr.ISVALIDREF_inSz                  := ISVALIDREF_inSz;
          str_Kr.ISVALIDREF_inDp                  := ISVALIDREF_inDp;
          str_Kr.continueHoldCommand              := continueHoldCommand;

          data_Ini:=False;
          Init := TRUE;
     END_IF;
   IF Init THEN
          ISVALIDREF_statOn:= false;
          ISVALIDREF_statOff:= false;
          ISVALIDREF_cmdOn:= false;
          ISVALIDREF_cmdOff:= false;
          ISVALIDREF_inSo:= false;
          ISVALIDREF_inSz:= false;
          ISVALIDREF_inDp:= false;
          continueHoldCommand:= T#0S;
    END_IF;
END_FUNCTION_BLOCK

FUNCTION_BLOCK fb_AiSourceMlp
  VAR_INPUT
    arAIN : TItemAIN;
    err_mod : TItemDIN;
  END_VAR
  VAR_IN_OUT
    strAI : struct_AI;
  END_VAR
  VAR
    _statusAi : TYPE_StatusAi;
    _commandAnalog : TYPE_CommandAnalog;
    _sunpackerCommand : fb_sunpackerCommand;
    _AnalogLimitFlags : TYPE_AnalogLimitFlags;
    notReliable : BOOL;
    _lastValue : LREAL;
    resetCmdTimer : TON;
    _LastValueTimer : TON;
    resetCmdTimerPriznak : BOOL;
    k : LREAL;
    b : LREAL;
    ap : LREAL;
    raznitsa : LREAL;
    rABS : LREAL;
    h : LREAL;
    mismatch : LREAL;
    parametr : BYTE;
    source : BYTE;
    cmd : BYTE;
    lastCmd : BYTE;
    source_for_Status : BYTE;
    cmd_for_Status : BYTE;
    command_error_for_Status : BYTE;
    onInit : BOOL;
    off_trig : R_TRIG;
    on_trig : R_TRIG;
    remont_trig : R_TRIG;
    LL_trig : R_TRIG;
    HL_trig : R_TRIG;
    Normal_trig : R_TRIG;
    Nedostover_trig : R_TRIG;
  END_VAR

  strAI.opcCommandsDisabled := strAI.inopcCommandsDisabled ;

  (* ---- При первом пуске принимаем значение уставок ---- *)
  IF NOT onInit THEN

            strAI.LL := strAI.dLL;
            strAI.HL := strAI.dHL;

            strAI.MaxChangeSpeed     := strAI.dMaxChangeSpeed;
            strAI.MaxChangeSpeedDown := strAI.dMaxChangeSpeedDown;

            IF strAI.ISVALIDREF_HA THEN strAI.HA := strAI.dHA; END_IF;

            IF strAI.ISVALIDREF_LA THEN strAI.LA := strAI.dLA; END_IF;

            IF strAI.ISVALIDREF_HW THEN strAI.HW := strAI.dHW; END_IF;

            IF strAI.ISVALIDREF_LW THEN strAI.LW := strAI.dLW; END_IF;

  	onInit  := TRUE;
  END_IF;

  (* ---- пересчет тока в физ величину ---- *)
  k := (strAI.HL - strAI.LL)/(strAI.inpHl - strAI.inpLL);
  b := strAI.LL - k * strAI.inpLL;
  strAI.value := k * arAIN.dblValue + b;

  (* ---- определение обрыва и кз ----- *)

  strAI.blConnect :=(*(UINT_TO_WORD(arAIN.wFlags) = 1472) and*) (UINT_TO_WORD(err_mod.wValue) = 20) and (UINT_TO_WORD(err_mod.wFlags) = 192);
  IF NOT strAI.blConnect THEN
      strAI.interval := _statusAi.NOTDEFINED;
  ELSIF ((arAIN.dblValue < strAI.currentBreakCircuit) AND (strAI.currentBreakCircuit > 0.0)) OR ((strAI.interval = _statusAi.LL) AND (arAIN.dblValue < (strAI.currentBreakCircuit + 100.0))) THEN
      strAI.interval := _statusAi.LL;
  ELSIF ((arAIN.dblValue > strAI.currentShotCircuit) AND (strAI.currentShotCircuit > 0.0)) OR ((strAI.interval = _statusAi.HL) AND (arAIN.dblValue > (strAI.currentShotCircuit - 100.0))) THEN
      strAI.interval := _statusAi.HL;
  ELSE
      strAI.interval := _statusAi.normal;
  END_IF;

  IF NOT strAI.imit THEN
  	(* Расчет апертурного фильтра*)
  	ap := strAI.aperturFilter * 0.01 * (strAI.HL - strAI.LL);
  	IF strAI.aperturFilter <> 0.0 THEN raznitsa := strAI.value- _lastValue;
  		IF 	raznitsa < 0.0 	THEN 	rABS := -raznitsa; 		ELSE 	rABS := raznitsa; 		END_IF;
  		IF 	rABS > ap 	THEN 	strAI.value := strAI.value;	ELSE 	strAI.value := _lastValue; 	END_IF;
  	END_IF;

  	(* Расчет экпоненциального фильтра*)
  	IF strAI.exponentialFilter <> 0.0 THEN strAI.value := (strAI.exponentialFilter * strAI.value) + ((1.0 - strAI.exponentialFilter) * _lastValue); END_IF;
  ELSE
  	strAI.interval := _statusAi.normal;
  END_IF;

  IF notReliable THEN strAI.interval := _statusAi.NOTRELIABLE; END_IF;

  IF NOT notReliable THEN
  	IF strAI.interval >= _statusAi.normal THEN
  		strAI.interval := _statusAi.NOTDEFINED;
  		h := strAI.histeresis* 0.01 * (strAI.HL-strAI.LL);
  		(*определение выхода за аппаратные границы вынесено в GetData.здесь только для нужд имитации*)
  		IF strAI.imit THEN
  			mismatch := strAI.rassoglasovanie * 0.01 * (strAI.HL - strAI.LL);
  			IF ( strAI.value < strAI.LL - mismatch)   THEN strAI.interval := _statusAi.LL;
  			ELSIF  (strAI.value > strAI.Hl + mismatch) THEN strAI.interval := _statusAi.HL; END_IF;
  		ELSE
  			strAI.interval := _statusAi.normal;
  			IF strAI.ISVALIDREF_LA AND NOT strAI.Disabled_LA AND (strAI.interval = _statusAi.normal) THEN
  				IF (strAI.value  < strAI.LA) OR ((strAI.interval = _statusAi.LA)  AND ((strAI.value - h) < strAI.LA))  THEN
  					strAI.interval := _statusAi.LA;
  				END_IF;
  			END_IF;
  			IF strAI.ISVALIDREF_HA  AND NOT strAI.Disabled_HA AND (strAI.interval = _statusAi.normal)  THEN
  				IF (strAI.value > strAI.HA) OR ((strAI.interval = _statusAi.HA)  AND ((strAI.value + h) > strAI.HA))  THEN
  					strAI.interval := _statusAi.HA;
  				END_IF;
  			END_IF;
  			IF strAI.ISVALIDREF_LW AND NOT strAI.Disabled_LW AND (strAI.interval = _statusAi.normal)  THEN
  				IF (strAI.value < strAI.LW) OR ((strAI.interval = _statusAi.LW)  AND ((strAI.value - h) < strAI.LW)) THEN
  					strAI.interval := _statusAi.LW;
  				END_IF;
  			END_IF;
  			IF strAI.ISVALIDREF_HW AND NOT strAI.Disabled_HW  AND (strAI.interval = _statusAi.normal) THEN
  				IF (strAI.value > strAI.HW)  OR ((strAI.interval = _statusAi.HW)  AND ((strAI.value + h) > strAI.HW))   THEN
  					strAI.interval := _statusAi.HW;
  				END_IF;
  			END_IF;
  		END_IF;
  	END_IF;
  ELSE
  	strAI.interval := _statusAi.NOTRELIABLE;
  END_IF;

  IF strAI.remont THEN strAI.interval := _statusAi.NOTDEFINED; END_IF;

  (* ---- Если управление с ВУ заблокировано, то  передаем команду из алгоритма ---- *)
  IF strAI.inOpcCommandsDisabled THEN
  	strAI.inCommand := strAI.inCommand_Alg;
  ELSE (* иначе передаем команду с АРМа*)
  	strAI.inCommand := strAI.inCommand_ARM;
  END_IF;

  _sunpackerCommand(command := strAI.inCommand);
  	source := _sunpackerCommand.source;
  	parametr := _sunpackerCommand.parametr;
  	cmd := _sunpackerCommand.cmd;

  IF cmd <> 0 AND lastCmd <> cmd and (((NOT strAI.opcCommandsDisabled) AND source > 0) OR source = 0) then
  	CASE BYTE_TO_INT(cmd) OF
  	(*cmd_SetUstavki*) 1 :
  				IF ((parametr AND _AnalogLimitFlags.LL) <> 0)		             	THEN 	strAI.LL := strAI.dLL; END_IF;
  				IF ((parametr AND _AnalogLimitFlags.HL) <> 0)		 	          THEN	strAI.HL := strAI.dHL; END_IF;
  				IF ((parametr AND _AnalogLimitFlags.LA) <> 0) AND strAI.ISVALIDREF_LA 	THEN	strAI.LA := strAI.dLA; END_IF;
  				IF ((parametr AND _AnalogLimitFlags.HA) <> 0) AND strAI.ISVALIDREF_HA 	THEN	strAI.HA := strAI.dHA; END_IF;
  				IF ((parametr AND _AnalogLimitFlags.LW) <> 0) AND strAI.ISVALIDREF_LW 	THEN	strAI.LW := strAI.dLW; END_IF;
  				IF ((parametr AND _AnalogLimitFlags.HW) <> 0) AND strAI.ISVALIDREF_HW 	THEN	strAI.HW := strAI.dHW; END_IF;
                                          IF ((parametr AND _AnalogLimitFlags.SipUP) <> 0)                       	THEN	strAI.MaxChangeSpeed     := strAI.dMaxChangeSpeed;     END_IF;
  				IF ((parametr AND _AnalogLimitFlags.SipDown) <> 0)                      	THEN	strAI.MaxChangeSpeedDown := strAI.dMaxChangeSpeedDown; END_IF;

  	(*cmd_SetRemont*) 6 :
  				strAI.remont := TRUE;
  	(*cmd_ResetRemont*) 7 :
  				strAI.remont := FALSE;
  	(*cmd_kvitNotReliable*) 4 :
  				notReliable := FALSE;
  	END_CASE;
  	source_for_Status := source;
  	cmd_for_Status := cmd;
  	command_error_for_Status := 0;
  	resetCmdTimer(IN := FALSE);
  	resetCmdTimerPriznak := TRUE;
  END_IF;
  lastCmd := cmd;

  resetCmdTimer(IN := resetCmdTimerPriznak, PT := T#5S);
  IF resetCmdTimer.Q THEN
  	resetCmdTimerPriznak := FALSE;
  	source_for_Status := 0;
  	cmd_for_Status := 0;
  	command_error_for_Status := 0;
  END_IF;

  strAI.NS_Min := (strAI.value < strAI.minValue) AND strAI.minValue_ISVALIDREF;
  strAI.NS_Max := (strAI.value > strAI.maxValue) AND strAI.maxValue_ISVALIDREF;

  strAI.NS := (strAI.interval <= _statusAi.normal) AND NOT strAI.remont;

  Normal_trig(CLK := strAI.interval >= _statusAi.normal);

  IF NOT Normal_trig.Q THEN
  	_LastValueTimer(PT := T#1S);
  	IF (strAI.value<>_lastValue) OR _LastValueTimer.Q THEN
  		IF (_LastValueTimer.ET>T#0MS) THEN
  			strAI.ChangeSpeed:=(strAI.value-_lastValue)/(TIME_TO_LREAL(_LastValueTimer.ET));
  		END_IF;
  		_LastValueTimer(IN:=FALSE);

  		_LastValueTimer(IN:=TRUE);
  	END_IF;
  END_IF;
  _lastValue := strAI.value;

  IF ((strAI.maxChangeSpeed<>0.0) OR  (strAI.maxChangeSpeedDown<>0.0)) AND ( strAI.interval>=_statusAi.normal) THEN
  		IF (strAI.ChangeSpeed>0.0) THEN
  		    IF (strAI.ChangeSpeed > strAI.maxChangeSpeed) AND (strAI.maxChangeSpeed>0.0000001) THEN
  			 notReliable:=TRUE;
  		    END_IF;
  		ELSE
  		    IF (ABS(strAI.ChangeSpeed)>strAI.maxChangeSpeedDown) AND (strAI.maxChangeSpeedDown>0.0000001)  THEN
                                 notReliable:=TRUE;
  		    END_IF;
  		END_IF;

  END_IF;

  strAI.status := SHL(BYTE_TO_DWORD(source_for_Status), 29) 		              (* Источник команды *)
  			OR SHL(BYTE_TO_DWORD(cmd_for_Status), 26) 	    (* Команда *)
  			OR SHL(BYTE_TO_DWORD(command_error_for_Status), 23)   (* Ошибка команды *)
  			OR SHL(BOOL_TO_DWORD(strAI.OpcCommandsDisabled ), 21) (* Управление в ВУ заблокировано *)
  			OR SHL(BOOL_TO_DWORD(strAI.Disabled_HA), 9)		    (* ВА исключена из формирования интервала *)
  			OR SHL(BOOL_TO_DWORD(strAI.Disabled_LA), 8)		    (* НА исключена из формирования интервала *)
  			OR SHL(BOOL_TO_DWORD(strAI.Disabled_HW), 7)		    (* ВП исключена из формирования интервала *)
  			OR SHL(BOOL_TO_DWORD(strAI.Disabled_LW), 6)	              (* НП исключена из формирования интервала *)
  			OR SHL(BOOL_TO_DWORD(strAI.NS), 5)			    (* неиспарвность сигнала *)
  			OR SHL(BOOL_TO_DWORD(strAI.remont), 4)	              (* Выведен в ремонт *)
  			OR BYTE_TO_DWORD(strAI.interval);	              (* интервал *)
END_FUNCTION_BLOCK

FUNCTION_BLOCK fb_AiProtection_Init
  VAR_INPUT
    data_Ini : BOOL;
    controlLimit : BYTE;
    delay : TIME;
    inTag : BYTE;
    inRunOnStart : BOOL;
  END_VAR
  VAR_IN_OUT
    str_AIp : struct_AiProtection;
  END_VAR
  VAR_OUTPUT
    Init : BOOL      := FALSE;
  END_VAR

  (*****            Функциональный блок переинициализации структуры  AiProtection          *****)

   Init := FALSE;

      IF data_Ini THEN                            (* Параметрам требуется переинициализация. *)
          str_AIp.controlLimit        := controlLimit;
          str_AIp.delay               := delay;
          str_AIp.inTag               := inTag;
          str_AIp.inRunOnStart        := inRunOnStart;

          data_Ini:=FALSE;
          Init := TRUE;
      END_IF;
      IF Init THEN
          controlLimit:= 0;
          delay:= T#0S;
          inTag:= 0;
          inRunOnStart:= FALSE;
      END_IF;
END_FUNCTION_BLOCK

FUNCTION impulseSO : BOOL
  VAR_IN_OUT
    so : struct_singleOutput;
  END_VAR
  VAR CONSTANT
    cmdImpulse : WORD      := 3;
  END_VAR

  IF NOT so.Q THEN
      so.inOpcCommandsDisabled:=TRUE;
      so.inCommand_Alg:=cmdImpulse;
  END_IF;
END_FUNCTION

FUNCTION_BLOCK SemiAutoPuskAlg
  VAR_IN_OUT
    StrAlg : struct_Alg;
  END_VAR
  VAR
    runOilsystem : struct_PhaseAlgoritm;
    runEngine : struct_PhaseAlgoritm;
    filling : struct_PhaseAlgoritm;
  END_VAR
  VAR_IN_OUT
    cmdRun1ph : struct_Question;
    cmdRun2ph : struct_Question;
    cmdRun3ph : struct_Question;
  END_VAR
  VAR
    fb_runOilsystem : fb_ph_algoritm;
    fb_runEngine : fb_ph_algoritm;
    fb_filling : fb_ph_algoritm;
    fb_cmdRun1ph : fb_Question;
    fb_cmdRun2ph : fb_Question;
    fb_cmdRun3ph : fb_Question;
    _sunpackerCommand : fb_sunpackerCommand;
    _PhaseAlgoritmAction : TYPE_PhaseAlgoritmAction;
    _statusDualInput : TYPE_statusDualInput;
    _Answers : TYPE_Answers;
    source : BYTE;
    cmd : BYTE;
    lastCmd : BYTE;
    source_for_Status : BYTE;
    cmd_for_Status : BYTE;
    command_error_for_Status : BYTE;
    resetCmdTimer : TON;
    resetCmdTimerPriznak : BOOL;
    onInit : BOOL;
    waitReset : TON;
  END_VAR
  VAR_EXTERNAL
    algoritms : AlgoritmsConfig;
    ModeGpa : TYPE_ModeGpa;
    algManager : struct_AlgoritmsManager;
    IM : ImConfig;
  END_VAR

  IF NOT onInit THEN
                 cmdRun1ph.AnswerVariants:=_Answers.ANS_YES;
           fb_runOilsystem(phaseNumber:=0, act:=_run, waitCompletion:=TRUE);
                 cmdRun2ph.AnswerVariants:=_Answers.ANS_YES;
              fb_runEngine(phaseNumber:=1, act:=_run, waitCompletion:=TRUE);
                 cmdRun3ph.AnswerVariants:=_Answers.ANS_YES;
                fb_filling(phaseNumber:=2, act:=_run, waitCompletion:=TRUE);

  onInit:=TRUE;
  END_IF;
              fb_cmdRun1ph(StrQ:=cmdRun1ph);
           fb_runOilsystem(StrPh:=runOilsystem, alg:=algoritms.puskOilSystem);
              fb_cmdRun2ph(StrQ:=cmdRun2ph);
              fb_runEngine(StrPh:=runEngine, alg:=algoritms.engineRun);
              fb_cmdRun3ph(StrQ:=cmdRun3ph);
                fb_filling(StrPh:=filling, alg:=algoritms.filling);

  StrAlg.CanRun := StrAlg.inCanRun;
  StrAlg.OpcCommandsDisabled := StrAlg.inOpcCommandsDisabled;

  IF StrAlg.isRuning THEN

      StrAlg.hasError := runOilsystem.error OR runEngine.error OR filling.error;

      IF cmdRun1ph.answer = _Answers.ANS_YES THEN
  	runPhase(runOilsystem);
            resetQuestion(cmdRun1ph);
      END_IF;

      IF runOilsystem.top AND NOT runEngine.start THEN
           askQuestion(cmdRun2ph);
      END_IF;

      IF cmdRun2ph.answer = _Answers.ANS_YES THEN
           runPhase(runEngine);
           resetQuestion(cmdRun2ph);
      END_IF;

      IF runEngine.top AND NOT filling.start THEN
           askQuestion(cmdRun3ph);
      END_IF;

      IF cmdRun3ph.answer = _Answers.ANS_YES THEN
           runPhase(filling);
           resetQuestion(cmdRun3ph);
      END_IF;

      IF filling.top THEN
            waitReset(IN:=TRUE, PT:= T#2S);
      END_IF;

      IF waitReset.Q THEN

          IF Im.kran6.onStatus = _statusDualInput.STATUS_On THEN
  	algManager.nMode:= ModeGpa.MODE_WORK_Ring;
          END_IF;
          IF Im.kran6.onStatus = _statusDualInput.STATUS_Off THEN
  	algManager.nMode:= ModeGpa.MODE_WORK_Line;
          END_IF;

          resetIfRunning(StrAlg);
      END_IF;

      StrAlg.isEnded:= filling.top;

  END_IF;

  StrAlg.CanRun := StrAlg.inCanRun;
  StrAlg.OpcCommandsDisabled := StrAlg.inOpcCommandsDisabled;

  (* ---- Если управление с ВУ заблокировано, то  передаем команду из алгоритма ---- *)
  IF StrAlg.inOpcCommandsDisabled THEN
  	StrAlg.inCommand := StrAlg.inCommand_Alg;
  ELSE (* иначе передаем команду с АРМа*)
  	StrAlg.inCommand := StrAlg.inCommand_ARM;
  END_IF;

  _sunpackerCommand(command := StrAlg.inCommand);
  	source := _sunpackerCommand.source;
  	cmd := _sunpackerCommand.cmd;

  IF cmd <> 0 AND lastCmd <> cmd AND (((NOT StrAlg.opcCommandsDisabled) AND source > 0) OR source = 0) then
  	CASE BYTE_TO_INT(cmd) OF
  		(*cmdRun*) 1: 	IF (StrAlg.CanRun) THEN
  					StrAlg.isRuning := TRUE;
  					StrAlg.isEnded := FALSE;
  					StrAlg.hasError := FALSE;
  					(*****************       OnRun       *****************)

                                                    algoritms.puskOilSystem.inCanRun:= TRUE	;
                                                    algoritms.filling.inCanRun:= TRUE	;
                                                    algoritms.engineRun.inCanRun:= TRUE	;

                                                    algManager.nMode:=ModeGpa.MODE_MPUSK;
                                                    (*impulseSO(Im.SingleOutputs.VzvodBREO);*)
                                                    askQuestion(cmdRun1ph);

  					cmd_for_Status := cmd;
  					source_for_Status := source;
  					command_error_for_Status := 0;
  				ELSE
  					StrAlg.isRuning := FALSE;
  					StrAlg.isEnded := FALSE;
  					StrAlg.hasError 	:= FALSE;

  					cmd_for_Status := 0;
  					source_for_Status := source;
  					command_error_for_Status := cmd;
  				END_IF;
  		(*cmdReset*) 2: 	StrAlg.isRuning := FALSE;
  				StrAlg.isEnded := FALSE;
  				StrAlg.hasError 	:= FALSE;

                                           (*****************       OnReset       *****************)
                                          waitReset(IN:=FALSE);
                                          StrAlg.inCanRun:=FALSE;

                                          resetPhase(runOilsystem);
                                          resetPhase(runEngine);
                                          resetPhase(filling);

                                          resetQuestion(cmdRun1ph);
                                          resetQuestion(cmdRun2ph);
                                          resetQuestion(cmdRun3ph);

                                          StrAlg.inOpcCommandsDisabled:=FALSE;

  				cmd_for_Status := cmd;
  				source_for_Status := source;
  				command_error_for_Status := 0;
  	END_CASE;
  	resetCmdTimer(IN := false);
  	resetCmdTimerPriznak := TRUE;
  END_IF;
  lastCmd := cmd;

  resetCmdTimer(IN := resetCmdTimerPriznak, PT := T#5S);
  IF resetCmdTimer.Q THEN
  	resetCmdTimerPriznak := FALSE;
  	source_for_Status := 0;
  	cmd_for_Status := 0;
  	command_error_for_Status := 0;
  END_IF;

  StrAlg.Start:= runOilsystem.startStatus
              OR runEngine.startStatus
              OR filling.startStatus;

  StrAlg.Error:= runOilsystem.errorStatus
              OR runEngine.errorStatus
              OR filling.errorStatus;

  StrAlg.Top:=   runOilsystem.topStatus
              OR runEngine.topStatus
              OR filling.topStatus;

  (*TODO: TYPE PROGRAM CODE HERE*)
  StrAlg.status :=  SHL(BYTE_TO_DWORD(source_for_Status), 29)
  			OR SHL(BYTE_TO_DWORD(cmd_for_Status), 26)
  			OR SHL(BYTE_TO_DWORD(command_error_for_Status), 23)
  			OR SHL(BOOL_TO_DWORD(StrAlg.OpcCommandsDisabled ), 21)
  			OR SHL(BOOL_TO_DWORD(StrAlg.hasError),4)
  			OR SHL(BOOL_TO_DWORD(StrAlg.CanRun),2)
  			OR SHL(BOOL_TO_DWORD(StrAlg.isEnded),1)
  			OR BOOL_TO_DWORD(StrAlg.isRuning);
END_FUNCTION_BLOCK

FUNCTION resetAllProtections : BOOL
  VAR_IN_OUT
    protections : ProtectionsConfig;
  END_VAR

  resetAiProtection(protections.Topornogo_podshipnika_EDT_1);
  resetAiProtection(protections.Toy_podshipnika_EDT_2);
  resetAiProtection(protections.Toy_podshipnika_kol_EDT_3);
  resetAiProtection(protections.Toy_podshipnika_kol_EDT_4);
  resetAiProtection(protections.To_podshipnika_shest_red_EDT_5);
  resetAiProtection(protections.To_podshipnika_shest_red_EDT_6);
  resetAiProtection(protections.To_podshipnika_N_EDT_7);
  resetAiProtection(protections.To_podshipnika_svob_konca_EDT_8);
  resetAiProtection(protections.Ty_podshipnika_rab_kol_EDT_9);
  resetAiProtection(protections.Typornogo_podshipnika_nerab_kolodok_HT_10);
  resetAiProtection(protections.Tgaza_na_vyhode_H);
  resetAiProtection(protections.Os_sdvig_nagnetatelja_plus);
  resetAiProtection(protections.Os_sdvig_nagnetatelja_minus);
  resetAiProtection(protections.Pgaza_na_vyhode_nagnetatelia_GPA_STOP);
  resetAiProtection(protections.Pgaza_na_vhode_nagnetatelia_GPA_STOP);
  resetAiProtection(protections.Pgaza_na_vyhode_nagnetatelia);
  resetAiProtection(protections.dPmaslo_gaz);
  resetAiProtection(protections.Pmaslo_sm_nizkoe);
  resetAiProtection(protections.Pmaslo_sm_vysokoe);
  resetAiProtection(protections.Vibro_skorost_OPED_T1);
  resetAiProtection(protections.Vibro_skorost_OPED_T2);
  resetAiProtection(protections.Vibro_skorost_OYP_kolesa_ED_T3);
  resetAiProtection(protections.Vibro_skorost_OP_kolesa_RH_T4);
  resetAiProtection(protections.Vibro_skorost_OP_shesterni_RED_T5);
  resetAiProtection(protections.Vibro_skorost_OP_shesterni_RED_T6);

  resetDiProtection(protections.dPmaslo_gaz_less100);
  resetDiProtection(protections.Reg_vozb_off);
  resetDiProtection(protections.Fail_chastotnii_pusk);
  resetDiProtection(protections.Off_avar_vikluchatel);
  resetDiProtection(protections.AOKC_SHKC);
  resetDiProtection(protections.AO_PRU);
  resetDiProtection(protections.AO_ot_SHU);
  resetDiProtection(protections.mvOff);
  resetDiProtection(protections.Kran1_sdvig);
  resetDiProtection(protections.Reg_vozb_off);
  resetDiProtection(protections.Kran2_sdvig);
END_FUNCTION

FUNCTION UnBlockAllIM : BOOL
  VAR_IN_OUT
    IM : ImConfig;
  END_VAR

  (*IF IM.TypeSwitch.Value = 1 THEN*)

  IF IM.Kran1.inOpcCommandsDisabled   THEN IM.Kran1.inOpcCommandsDisabled:=FALSE; END_IF;
  IF IM.Kran2.inOpcCommandsDisabled   THEN IM.Kran2.inOpcCommandsDisabled:=FALSE; END_IF;
  IF IM.Kran3b.inOpcCommandsDisabled  THEN IM.Kran3b.inOpcCommandsDisabled:=FALSE; END_IF;
  IF IM.Kran4.inOpcCommandsDisabled   THEN IM.Kran4.inOpcCommandsDisabled:=FALSE; END_IF;
  IF IM.Kran5.inOpcCommandsDisabled   THEN IM.Kran5.inOpcCommandsDisabled:=FALSE; END_IF;
  (*IF IM.Kran6.inOpcCommandsDisabled   THEN IM.Kran6.inOpcCommandsDisabled:=FALSE; END_IF;*)
  (*END_IF;*)

  IF IM.nu1.inOpcCommandsDisabled     THEN IM.nu1.inOpcCommandsDisabled:=FALSE; END_IF;
  IF IM.nu2.inOpcCommandsDisabled     THEN IM.nu2.inOpcCommandsDisabled:=FALSE; END_IF;
  IF IM.pns.inOpcCommandsDisabled     THEN IM.pns.inOpcCommandsDisabled:=FALSE; END_IF;
  IF IM.v1_Avom.inOpcCommandsDisabled THEN IM.v1_Avom.inOpcCommandsDisabled:=FALSE; END_IF;
  IF IM.v2_Avom.inOpcCommandsDisabled THEN IM.v2_Avom.inOpcCommandsDisabled:=FALSE; END_IF;
  (*IF IM.Ten.inOpcCommandsDisabled     THEN IM.Ten.inOpcCommandsDisabled:=FALSE; END_IF;*)
  IF IM.mv.inOpcCommandsDisabled      THEN IM.mv.inOpcCommandsDisabled:=FALSE; END_IF;
END_FUNCTION

FUNCTION BlockAllIM : BOOL
  VAR_IN_OUT
    IM : ImConfig;
  END_VAR

  IF NOT IM.Kran1.inOpcCommandsDisabled   THEN IM.Kran1.inOpcCommandsDisabled:=TRUE; END_IF;
  IF NOT IM.Kran2.inOpcCommandsDisabled   THEN IM.Kran2.inOpcCommandsDisabled:=TRUE; END_IF;
  IF NOT IM.Kran3b.inOpcCommandsDisabled  THEN IM.Kran3b.inOpcCommandsDisabled:=TRUE; END_IF;
  IF NOT IM.Kran4.inOpcCommandsDisabled   THEN IM.Kran4.inOpcCommandsDisabled:=TRUE; END_IF;
  IF NOT IM.Kran5.inOpcCommandsDisabled   THEN IM.Kran5.inOpcCommandsDisabled:=TRUE; END_IF;
  (*IF NOT IM.Kran6.inOpcCommandsDisabled   THEN IM.Kran6.inOpcCommandsDisabled:=TRUE; END_IF;*)

  IF NOT IM.nu1.inOpcCommandsDisabled     THEN IM.nu1.inOpcCommandsDisabled:=TRUE; END_IF;
  IF NOT IM.nu2.inOpcCommandsDisabled     THEN IM.nu2.inOpcCommandsDisabled:=TRUE; END_IF;
  IF NOT IM.pns.inOpcCommandsDisabled     THEN IM.pns.inOpcCommandsDisabled:=TRUE; END_IF;
  IF NOT IM.v1_Avom.inOpcCommandsDisabled THEN IM.v1_Avom.inOpcCommandsDisabled:=TRUE; END_IF;
  IF NOT IM.v2_Avom.inOpcCommandsDisabled THEN IM.v2_Avom.inOpcCommandsDisabled:=TRUE; END_IF;
  (*IF NOT IM.Ten.inOpcCommandsDisabled     THEN IM.Ten.inOpcCommandsDisabled:=TRUE; END_IF;*)
  IF NOT IM.mv.inOpcCommandsDisabled      THEN IM.mv.inOpcCommandsDisabled:=TRUE; END_IF;
END_FUNCTION

FUNCTION_BLOCK RemontAlg
  VAR_IN_OUT
    StrAlg : struct_Alg;
  END_VAR
  VAR
    _sunpackerCommand : fb_sunpackerCommand;
    source : BYTE;
    cmd : BYTE;
    lastCmd : BYTE;
    source_for_Status : BYTE;
    cmd_for_Status : BYTE;
    command_error_for_Status : BYTE;
    resetCmdTimer : TON;
    resetCmdTimerPriznak : BOOL;
  END_VAR
  VAR_EXTERNAL
    protectManager : struct_ProtectionsManager;
    algManager : struct_AlgoritmsManager;
    ModeGpa : TYPE_ModeGpa;
    PMcommand : TYPE_CommandsPotectionsManager;
    IM : ImConfig;
  END_VAR

  StrAlg.CanRun := StrAlg.inCanRun;
  StrAlg.OpcCommandsDisabled := StrAlg.inOpcCommandsDisabled;

  (* ---- Если управление с ВУ заблокировано, то передаем команду из алгоритма ---- *)
  IF StrAlg.inOpcCommandsDisabled THEN
  	StrAlg.inCommand := StrAlg.inCommand_Alg;
  ELSE (* иначе передаем команду с АРМа*)
  	StrAlg.inCommand := StrAlg.inCommand_ARM;
  END_IF;

  _sunpackerCommand(command := StrAlg.inCommand);
  	source := _sunpackerCommand.source;
  	cmd := _sunpackerCommand.cmd;

  IF cmd <> 0 AND lastCmd <> cmd AND (((NOT StrAlg.opcCommandsDisabled) AND source > 0) OR source = 0) then
  	CASE BYTE_TO_INT(cmd) OF
  		(*cmdRun*) 1: 	IF (StrAlg.CanRun) THEN
  					StrAlg.isRuning := TRUE;
  					StrAlg.isEnded := FALSE;
  					StrAlg.hasError 	:= FALSE;
                                               (*****************       OnRun       *****************)
                                                        algManager.nMode:=ModeGpa.MODE_REMONT;
                                                        protectManager.inCommand:=PMcommand.ResetAllProtections;
  					    UnBlockAllIM(IM);
                                                    (*StrAlg.inOpcCommandsDisabled:=FALSE;*)
  					cmd_for_Status := cmd;
  					source_for_Status := source;
  					command_error_for_Status := 0;
  				ELSE
  					StrAlg.isRuning := FALSE;
  					StrAlg.isEnded := FALSE;
  					StrAlg.hasError 	:= FALSE;

  					cmd_for_Status := 0;
  					source_for_Status := source;
  					command_error_for_Status := cmd;
  				END_IF;
  		(*cmdReset*) 2: 	StrAlg.isRuning := FALSE;
  				StrAlg.isEnded := FALSE;
  				StrAlg.hasError 	:= FALSE;
                                          (*****************       OnReset       *****************)
                                                    BlockAllIM(IM);
                                                    protectManager.inCommand:=PMcommand.RestartAllProtections;
                                                    algManager.nMode:=ModeGpa.MODE_STOP;

  				cmd_for_Status := cmd;
  				source_for_Status := source;
  				command_error_for_Status := 0;
  	END_CASE;
  	resetCmdTimer(IN := false);
  	resetCmdTimerPriznak := TRUE;
  END_IF;
  lastCmd := cmd;

  resetCmdTimer(IN := resetCmdTimerPriznak, PT := T#5S);
  IF resetCmdTimer.Q THEN
  	resetCmdTimerPriznak := FALSE;
  	source_for_Status := 0;
  	cmd_for_Status := 0;
  	command_error_for_Status := 0;
  END_IF;

  StrAlg.status :=  SHL(BYTE_TO_DWORD(source_for_Status), 29)
  			OR SHL(BYTE_TO_DWORD(cmd_for_Status), 26)
  			OR SHL(BYTE_TO_DWORD(command_error_for_Status), 23)
  			OR SHL(BOOL_TO_DWORD(StrAlg.OpcCommandsDisabled ), 21)
  			OR SHL(BOOL_TO_DWORD(StrAlg.hasError),4)
  			OR SHL(BOOL_TO_DWORD(StrAlg.CanRun),2)
  			OR SHL(BOOL_TO_DWORD(StrAlg.isEnded),1)
  			OR BOOL_TO_DWORD(StrAlg.isRuning);
END_FUNCTION_BLOCK

FUNCTION_BLOCK Pusk_third_faza
  VAR_IN_OUT
    StrAlg : struct_Alg;
  END_VAR
  VAR
    timer480 : struct_PhaseAlgoritm;
    kran4Open : struct_PhaseAlgoritm;
    waitAfterKran4 : struct_PhaseAlgoritm;
    kran5Close : struct_PhaseAlgoritm;
    kran3bOpen : struct_PhaseAlgoritm;
    dP_kr1less100 : struct_PhaseAlgoritm;
    Pvh_vyhMore5 : struct_PhaseAlgoritm;
    kran1Open : struct_PhaseAlgoritm;
    kran2Open : struct_PhaseAlgoritm;
    kran3Open : struct_PhaseAlgoritm;
    kran3bClose : struct_PhaseAlgoritm;
    Err_ALG : struct_PhaseAlgoritm;
    fb_timer480 : fb_ph_Timer;
    fb_kran4Open : fb_ph_Kran;
    fb_waitAfterKran4 : fb_ph_Timer;
    fb_kran5Close : fb_ph_Kran;
    fb_kran3bOpen : fb_ph_Kran;
    fb_dP_kr1less100 : fb_ph_algoritm;
    fb_Pvh_vyhMore5 : fb_ph_algoritm;
    fb_kran1Open : fb_ph_Kran;
    fb_kran2Open : fb_ph_Kran;
    fb_kran3Open : fb_ph_Kran;
    fb_kran3bClose : fb_ph_Kran;
    fb_Err_ALG : fb_ph_algoritm;
    _sunpackerCommand : fb_sunpackerCommand;
    _statusDualInput : TYPE_statusDualInput;
    _Answers : TYPE_Answers;
    source : BYTE;
    cmd : BYTE;
    lastCmd : BYTE;
    source_for_Status : BYTE;
    cmd_for_Status : BYTE;
    command_error_for_Status : BYTE;
    resetCmdTimer : TON;
    resetCmdTimerPriznak : BOOL;
    onInit : BOOL;
    waitReset : TON;
  END_VAR
  VAR_EXTERNAL
    ModeGpa : TYPE_ModeGpa;
    algManager : struct_AlgoritmsManager;
    IM : ImConfig;
    protections : ProtectionsConfig;
    algoritms : AlgoritmsConfig;
    ai : AiConfig;
  END_VAR
  VAR
    statusAi : TYPE_StatusAi;
  END_VAR
